# B&R Automation Studio project TD52 (part 133)

#### MsgSA.var
```iecst
VAR
	iAdrAmmBase2MM : UDINT;
	iAdrMM2AmmBase : UDINT;
	xMsg2214 : Msg;
	xMsg2254 : Msg;
	xMsg2255 : Msg;
	xMsg2256 : Msg;
	xMsg2281 : Msg;
	xMsg2297 : Msg;
	xMsg2298 : Msg;
	xMsg2299 : Msg; (* alarm for cylinder pressure sensor saturation*)
	xMsg9318 : Msg; (* warning for cylinder pressure sensor saturation*)
	xMsg2585 : Msg;
	xMsg2800 : Msg;
	xMsg2816 : Msg;
	xMsg2817 : Msg;
	xMsg2818 : Msg;
	xMsg2819 : Msg;
	xMsg2820 : Msg;
	xMsg2898 : Msg;
	xMsg2906 : Msg;
	xMsg2907 : Msg;
	xMsg3270 : Msg;
	xMsg3271 : Msg;
	xMsg3272 : Msg;
	xMsg3273 : Msg;
	xMsg3275 : Msg;
	xMsg3276 : Msg;
	xMsg3277 : Msg;
	xMsg3278 : Msg;
	xMsg3283 : Msg;
	xMsg3284 : Msg;
	xMsg3286 : Msg;
	xMsg3287 : Msg;
	xMsg3288 : Msg;
	xMsg3291 : Msg;
	xMsg3292 : Msg;
	xMsg3293 : Msg;
	xMsg3294 : Msg;
	xMsg3330 : Msg;
	xMsg3331 : Msg;
	xMsg3332 : Msg;
	xMsg3333 : Msg;
	xMsg3334 : Msg;
	xMsg3335 : Msg;
	xMsg3336 : Msg;
	xMsg3337 : Msg;
	xMsg3338 : Msg;
	xMsg3343 : Msg;
	xMsg3344 : Msg;
	xMsg3345 : Msg;
	xMsg3530 : Msg;
	xMsg3531 : Msg;
	xMsg3533 : Msg;
	xMsg3535 : Msg;
	xMsg3536 : Msg;
	xMsg3537 : Msg;
	xMsg3539 : Msg;
	xMsg3544 : Msg;
	xMsg3545 : Msg;
	xMsg3546 : Msg;
	xMsg3547 : Msg;
	xMsg3548 : Msg;
	xMsg3549 : Msg;
	xMsg3550 : Msg;
	xMsg3551 : Msg;
	xMsg3552 : Msg;
	xMsg3553 : Msg;
	xMsg3554 : Msg;
	xMsg2910 : Msg;
	xMsg2476 : Msg;
	xMsg2334 : Msg;
	xMsg9027 : Msg;
	xMsg2335 : Msg;
	xMsg9028 : Msg;
	xMsg9320 : Msg;
	xMsg9045 : Msg;
	xMsg9321 : Msg;
	xMsg9046 : Msg;
	xMsg2493 : Msg;
	xMsg2939 : Msg;
	xMsg9066 : Msg;
	xMsg9050 : Msg;
	xMsg9350 : Msg;
END_VAR
```


### Package Logical/Synchronization - SY: Synchronization

### Data object Logical/Synchronization/META_SY (Simple) - MODUL META data file

#### META_SY.dat
```
; *******************************************************************************
; AGGR: Module Meta Data (data module)
;
; This code is confidential and proprietary to the INNIO Company.
; It may not be used in any form, or reproduced in any manner, without the express
; written permission of the INNIO Company.
; Copyright, INNIO Company, 2022
;
; Customized modifications: -
; ------------------------
;
; History:
; -------
; V03.99.00.00	06.03.2013	Weitzer, 	generated for modular software
;				02.10.2013	lettenb.	descriptions setted
;				04.12.2013	lettenb.	dependencies added
; V04.00.00.00	31.01.2014	lettenb.	version + dependencies changed
; V04.00.03.00	22.07.2014	lettenb.	para_task update
; V04.03.00.00	02.03.2015	lettenb.	version + dependencies changed (920)
; V04.03.00.00	11.06.2015	Zengerer 	version + dependencies changed (IF change with array index 0 for compatibility with c-tasks)
;				15.06.2015  lettenb.	PARAMETER_CHK expanded
; V04.04.00.00	04.07.2016	lettenb.	version changed
;               20.03.2017  lettenb.	fast detection of freq.changes, dyn.gridcode III
; V04.05.00.00	11.12.2017	lettenb.	gridcode logic added
; V04.05.01.00	09.03.2018	Perktold	delayed A1042 trip (only HiHi part), 100ms normal, 500ms when LVRT Event is detected (for 5s)
;               18.09.2018	lettenb.	gcb IO monitoring, sequential arrangement changed, bu
; V04.06.00.00	21.09.2018  Perktold,   MsgSY: A1042 implemented 110% overload step 3s delay excluded bBDC_Emergency_OFF
; V04.07.00.00	11.12.2017	lettenb.	dataitems for diagnosis added
;				03.10.2019	lettenb.	perm data writing to CF 10s -> 10m, bu01
; V04.09.00.00	17.10.2019	lettenb.	gcbTC1, gcb closing time monitoring added
;				01.10.2020	lettenb.	OUT_SY.bMCB_DemSy, mcb controlled by customer, bugfix(heim, Referenzanlage AB85), bu02
; V04.10.00.00	16.10.2020  Weitzer		IN_SY.bCust_Dem_Sy added to GCB demand sy, IN_SY.bCust_Dem_RSy added to ton_mcb_dmnd_sy ELSE part
; V04.11.00.00	24.06.2021	Arnold		Open GCB in island on underfrequency IN_SY.bGCB_DCon_EC
;				07.07.2021	lettenb.	init xMsg2692.Num: 2693->2692, bugfix
; V04.12.00.00	02.05.2022	Schmidt		W2688 (high sync current) threshold increased from 50% to 75% of nominal current
;				29.06.2022	lettenb.	dead bb synch added
; V04.13.00.00  26.09.2023	Farre,		LCB operating message when open (B9083) or closed (B9084)
;				14.11.2023	Hohensinner	Added LV_GCB task (Modbus RTU connection to LV GCBs)
;				20.11.2023	Farre,		added "bypass MCB" and "request power mode" interfaces from CU needed for Microgrid (2023-168)
;				29.11.2023	Goenczi,	Standardization changes (Aggreko)
;				22.01.2024	Astner		Added iModule to OUT_SY
; V04.14.00.00	25.10.2024	Farre,		GCB Opening Failure - W1217 and reverse power connected to GCB_OpF command (2024-241)
;				22.11.2024	Fahringer	Use generator current before GCB closure to check 2% change (2024-238)
;										GCB closing time monitoring for more than 40ms (2024-238)
;				22.11.2024	Farre		bMMD_SyncDO only when used for GCB (2024-238)
;
; Instructions for use:
; --------------------
; make only changes at the version numbers
;
; Outstandings:
; ------------
;
; *******************************************************************************
;
"<META>"
;
; Module ID
"<MODUL>SY</MODUL>"
;
; Module Version (xx.yy.zz.cc)
"<VERSION>04.14.00.00</VERSION>"
;
; Module Basisupdate Version BU (00-99)
"<BASISUPDATE_VERSION>00</BASISUPDATE_VERSION>"
;
; Optional: specify order number for limitated module usage
"<ORDER></ORDER>" ;<!--(optional for restricted customizations; missing statement makes module valid for all orders)-->
;
; Parameter Check <PARAn Name='aAbcdef' MIN='xxx' MAX='yyy' />  (watch for correct spacings and apostrophs!)
"<PARAMETER_CHK>"
"<PARA1 Name='iEng_Motortype' MIN='208' MAX='920' />"
"<PARA2 Name='rN_EngStart_LimHi' MIN='50.0' MAX='2200.0' />"
"<PARA3 />"
"<PARA4 />"
"<PARA5 />"
"</PARAMETER_CHK>"
;
; Permanent Datamodule Filenames<!-- NAME ist ohne Dateiendung einzutragen; Nur für Counter und interne Parameter verwenden-->
"<DATAMODULES>" ;<!-- optional; mehrere DATAMODULES erlaubt-->
"	<DATAMODULE>par_SY</DATAMODULE>"
"	<DATAMODULE>perm_SY</DATAMODULE>"
"</DATAMODULES>"
;
; Dependencies Modules (MMxx.yy.zz.cc)
"<DEPENDENCIES>"
"	<DEPENDENCY MODULE='AB' VERSION='04.03.00.00' />"
"	<DEPENDENCY MODULE='CH' VERSION='04.00.00.00' />"
"	<DEPENDENCY MODULE='CU' VERSION='04.13.00.00' />"
"	<DEPENDENCY MODULE='EC' VERSION='04.06.00.00' />"
"	<DEPENDENCY MODULE='EG' VERSION='04.00.00.00' />"
"	<DEPENDENCY MODULE='GC' VERSION='04.14.00.00' />"
"	<DEPENDENCY MODULE='GR' VERSION='04.07.00.00' />"
"	<DEPENDENCY MODULE='GT' VERSION='04.00.00.00' />"
"	<DEPENDENCY MODULE='HA' VERSION='04.13.00.00' />"
"	<DEPENDENCY MODULE='HC' VERSION='04.07.00.00' />"
"	<DEPENDENCY MODULE='IG' VERSION='04.00.00.00' />"
"	<DEPENDENCY MODULE='OP' VERSION='04.13.00.00' />"
"	<DEPENDENCY MODULE='PB' VERSION='04.00.00.00' />"
"   <DEPENDENCY VISVERSION='02.14.00.00' />"			; Dependencies Visualization
"</DEPENDENCIES>"
;
; Module function description
"<MODULEFUNCTION>" ;<!-- short overview documentation of module function; add reference to detailed information, if available-->
"	<General>	"
"	Circuit breaker control. "
"	</General>	"
""
"	<F1 Name='Generator circuit breaker' LastModified='3.99.00.00'>"
"	Generator circuit breaker control and monitoring.	"
"	</F1>"
"	<F2 Name='Mains circuit breaker' LastModified='3.99.00.00'>"
"	Mains circuit breaker control and monitoring.	"
"	</F2>"
"	<F3 Name='Blackout start' LastModified='3.99.00.00'>"
"	Blackout start management.	"
"	</F3>"
"	<F4 Name='Load shedding' LastModified='3.99.00.00'>"
"	Load shedd management.	"
"	</F4>"
"	<F5 Name='Generator deexcitation' LastModified='3.99.00.00'>"
"	Generator deexcitation control.	"
"	</F5>"
"	<F6 Name='Synchronization alarm management' LastModified='4.04.00.00'>"
"	Synchronization alarm management.	"
"	</F6>"
"	<F7 Name='Mains monitoring' LastModified='4.04.00.00'>"
"	Mains monitoring (dyn.gridcode III)"
"	</F7>"
""
"	<Info>"
"   UPDATE V4.02.01	version + dependencies changed (IF change with array index 0 for compatibility with c-tasks)	"
"	</Info>"
""
"	<Customized LastModified='3.99.00.00'>"
"	- Nothing "
"	</Customized>	"
""
"</MODULEFUNCTION>"
;
"</META>"
```

### module_SY.typ
```iecst
TYPE
	IN_SY_struct : 	STRUCT
		tAB2SY : AmmBase2MM;
		tPB2MM : ParaBase2MM_type;
		iSt_OpMode : UDINT; (*status operation mode*) (*OldName:newPv; Cycle:5;*)
		iIdx_OMSS : INT; (*engine operation mode selection*) (*OldName:newPv; Cycle:5;*)
		rN_EngAct : REAL; (*engine speed actual [1/min]*) (*OldName:ANA.DREHZ; Cycle:5;*)
		bEng_RPSDem : BOOL; (*engine demanded *) (*OldName:A_AGFD; Cycle:5;*)
		bEng_Rdy_Aut_Exc : BOOL; (* engine ready for automatic operation *) (*OldName:BERAUT; Cycle:5;*)
		bGCB_Off_CNS : BOOL; (* generator circuit breaker opened by curent negative sequence *) (*OldName:gcb_off_iasy; Cycle:5;*)
		bGCB_Off_RP : BOOL; (* generator circuit breaker opened by reverse power *) (*OldName:gcb_off_rlsg; Cycle:5;*)
		bEng_Dem : BOOL; (* demand engine *) (*OldName:M_AGFD; Cycle:5;*)
		bEng_Dem_EPS : BOOL; (* engine demand for emergency operation *) (*OldName:M_NANF; Cycle:5;*)
		bGV_On : BOOL; (*Gas valves On *) (* OldName:M_GASV; Cyclic:5;*)
		rP_Nom : REAL; (* nominal power related to selected gas type [kW]*) (*OldName:PN_GASART[]; Cycle:5;*)
		bSCO_Active : BOOL; (* safety cut out gas valves glow ignition prevention *) (*OldName:SICH_SCHL; Cycle:5;*)
		rP_Act_Norm : REAL; (* actual power related to rP_Nom [%] *) (*OldName:P_IST_OF; Cycle:5;*)
		rP_Act_Norm_Filt : REAL; (* actual power related to rP_Nom filtered(1s) [%] *) (*OldName:P_IST; Cycle:5;*)
		bP_Red_Active : BOOL; (* power reduction active - any kind *) (*OldName:PredAkt; Cycle:5;*)
		bRelSy_Customized : BOOL; (*release synchronization from custom)*) (*OldName:newPv; Cycle:5;*)
		rP_MainsImport : REAL; (* mains import power [kW]*) (*OldName:Pmns_pv_1; Cycle:5;*)
		tEng_Run : HALioDo_Type; (* engine in operation *) (*OldName:BTRB; Cycle:5;*)
		tRel_Sync_Load : HALioDo_Type; (*DO release of sychronization and load*) (*OldName:SY_LFG; Cycle:5;*)
		tGrC_DCon : HALioDo_Type; (*DO: FALSE = Disconnect from Grid due to GridCode Event*) (* OldName: DO_GRIDCODE_DCON_TC1; Cycle:5; *)
		tTBMode : HALioDi_Type; (* DI test bench mode *) (*OldName:CIRCUITUS; Cycle:5;*)
		tBB_Alive : HALioDi_Type; (* DI bus bar alive *) (*OldName:DI_BB_ALIVE; Cycle:5;*)
		tBB_Dead_MMD : ARRAY[0..2]OF HALioDi_Type; (* DI bus bar dead from MMD *) (*OldName:DI_MMUSynchStatDO03; Cycle:5;*)
		tC_CB_EDC : HALioDi_Type; (* DI customer circuit breaker (engine) demand close *) (*OldName:DI_C_CB_EDC; Cycle:5;*)
		tC_CB_ESL : HALioDi_Type; (* DI customer circuit breaker (engine) status locked *) (*OldName:DI_C_CB_ESL; Cycle:5;*)
		tC_CB_Off : HALioDi_Type; (* DI customer circuit breaker opened *) (*OldName:DI_C_CB_OFF; Cycle:5;*)
		tC_CB_On : HALioDi_Type; (* DI customer circuit breaker closed *) (*OldName:DI_C_CB_ON; Cycle:5;*)
		tReq_PowMod : HALioDi_Type; (* DI request power operation mode *) (*OldName:DI_DMND_PM; Cycle:5;*)
		tEngDemIsland : HALioDi_Type; (* DI engine demand for island operation *) (*OldName:DI_ENG_DI; Cycle:5;*)
		tGCB_AGO : HALioDi_Type; (* DI all other generator circuit breaker off *) (*OldName:DI_GCB_AGO; Cycle:5;*)
		tGCB_DSY : HALioDi_Type; (* DI  generator circuit breaker demand synchronization (synchline) *) (*OldName:DI_GCB_DSY; Cycle:5;*)
		tGCB_DVM : HALioDi_Type; (* DI  generator circuit breaker demand voltage matching *) (*OldName:DI_GCB_DVM; Cycle:5;*)
		tGCB_MDL : HALioDi_Type; (* DI generator circuit breaker master demand lock (for closing other GCB to dead BB) *) (*OldName:DI_GCB_MDL; Cycle:5;*)
		tGCB_MRC : HALioDi_Type; (* DI generator circuit breaker master release close (to dead busbar) *) (*OldName:DI_GCB_MRC; Cycle:5;*)
		tGCB_OGP : HALioDi_Type; (* DI generator circuit breaker other generator parallel *) (*OldName:DI_GCB_OGP; Cycle:5;*)
		tGCB_On : HALioDi_Type; (* DI generator circuit breaker closed *) (*OldName:DI_GCB_ON; Cycle:5;*)
		tGCB_Rac : HALioDi_Type; (* DI generator circuit breaker racked in *) (*OldName:DI_GCB_RAC; Cycle:5;*)
		tGCB_Rdy : HALioDi_Type; (* DI generator circuit breaker ready (for close) *) (*OldName:DI_GCB_RDY; Cycle:5;*)
		tGCB_RI : HALioDi_Type; (* DI generator circuit breaker reelase island *) (*OldName:DI_GCB_RI; Cycle:5;*)
		tGCB_SM1 : HALioDi_Type; (* DI generator circuit breaker output signal monitoring 1 *) (*OldName:DI_GCB_SM1; Cycle:5;*)
		tGCB_SM2 : HALioDi_Type; (* DI generator circuit breaker contact signal monitoring 2 *) (*OldName:DI_GCB_SM2; Cycle:5;*)
		tGCB_Off : HALioDi_Type; (* DI generator circuit breaker opened *) (*OldName:DI_GCB_OFF; Cycle:5;*)
		tGCB_Earth : HALioDi_Type; (* DI generator circuit breaker position earth *) (*OldName:newPv; Cycle:5;*)
		tMCB_OL : HALioDi_Type; (* DI mains circuit breaker overload *) (*OldName:DI_MCB_OL; Cycle:5;*)
		tMCB_On : HALioDi_Type; (* DI mains circuit breaker closed *) (*OldName:DI_MCB_ON; Cycle:5;*)
		tMCB_Off : HALioDi_Type; (* DI mains circuit breaker opened *) (*OldName:DI_MCB_OFF; Cycle:5;*)
		tMCB_Rac : HALioDi_Type; (* DI mains circuit breaker racked in *) (*OldName:DI_MCB_RAC; Cycle:5;*)
		tMCB_Rdy : HALioDi_Type; (* DI mains circuit breaker ready (for close) *) (*OldName:DI_MCB_RDY; Cycle:5;*)
		tMCB_Rem : HALioDi_Type; (* DI mains circuit breaker remote (operating mode) *) (*OldName:DI_MCB_REM; Cycle:5;*)
		tMCB_SM : HALioDi_Type; (* DI mains circuit breaker signal monitoring *) (*OldName:DI_MCB_SM; Cycle:5;*)
		tMns_MDF : HALioDi_Type; (* DI mains monitoring device failure *) (*OldName:DI_MCB_MDF; Cycle:5;*)
		tMnsOk : HALioDi_Type; (* DI mains ok *) (*OldName:DI_MNS_OK; Cycle:5;*)
		tOnly_Island : HALioDi_Type; (* DI only island operation *) (*OldName:DI_ONLY_I; Cycle:5;*)
		tRel_BS : HALioDi_Type; (* DI release black start *) (*OldName:DI_REL_BS; Cycle:5;*)
		tRel_I : HALioDi_Type; (* DI release island operation *) (*OldName:DI_REL_I; Cycle:5;*)
		tRel_LS : HALioDi_Type; (* DI release load shedding *) (*OldName:DI_REL_LS; Cycle:5;*)
		tGCB_DRM : HALioDi_Type; (* DI generator circuit breaker demand MCB closing return to mains *) (*OldName:newPv; Cycle:5;*)
		tGen_RVM : HALioDi_Type; (* DI generator release voltage matching (leroy somer) *) (*OldName:newPv; Cycle:5;*)
		tSy_N_Up : HALioDi_Type; (* DI external speed matching UP *) (*OldName:newPv; Cycle:5;*)
		tSy_N_Down : HALioDi_Type; (* DI external speed matching DOWN *) (*OldName:newPv; Cycle:5;*)
		tLineCB_On : HALioDi_Type; (* DI line circuit breaker closed *) (*OldName:LIN_EIN; Cycle:5;*)
		tU_Avg : ARRAY[0..2]OF HALioAi_Type; (*AI generator voltage average value MMD [V]*) (*OldName:ANA.UDURCH; Cycle:5;*)
		tRelEngOpFromGSy : HALioDi_Type; (*DI release engine operation from 'gemeinsame'synchronization*) (*OldName:F_BLO; Cycle:5;*)
		tEarthCB_Off : HALioDi_Type; (*DI earth circuit breaker opened, france country specific*) (*OldName:DI_ECB_OFF; Cycle:5;*)
		tIsoCB_Off : HALioDi_Type; (*DI disconnecting circuit breaker opened, france country specific*) (*OldName:DI_ISOL; Cycle:5;*)
		tMnsOk_GTE : HALioDi_Type; (*DI mains ok GTE monitoring device, france country specific*) (*OldName:DI_GTE; Cycle:5;*)
		tMnsOk_TGS : HALioDi_Type; (*DI mains ok TGS monitoring device, france country specific*) (*OldName:DI_TGS; Cycle:5;*)
		tMnsOk_C13100 : HALioDi_Type; (*DI mains ok C13.100 monitoring device, france country specific*) (*OldName:DI_C13_100; Cycle:5;*)
		bMsg1026 : BOOL; (*engine shutdown failure *) (*OldName:M_ANSTAB; Cycle:5;*)
		bMsg1026_Test : BOOL; (*engine shutdown failure test*) (*OldName:newPv; Cycle:5;*)
		bMsg1134 : BOOL; (*Earth failure*) (*OldName:M_ERDS; Cycle:5;*)
		bMsg1036 : BOOL; (*overload short circuit*) (*OldName:M_ULKS; Cycle:5;*)
		bMsg1038 : BOOL; (*generator reverse power*) (*OldName:M_RLSG; Cycle:5;*)
		bMsg1073 : BOOL; (*generator over load from multi measuring device*) (*OldName:M_MMD_OL; Cycle:5;*)
		bMsg1132 : BOOL; (*generator differencial protection*) (*OldName:M_DIFF; Cycle:5;*)
		bMsg3319 : BOOL; (*generator protection trip*) (*OldName:M_GEN_PT; Cycle:5;*)
		rCust_SparePara : ARRAY[0..200]OF REAL; (*SPS_REZP1 to SPS_REZP200	*) (* OldName: SPS_REZP1, SPS_REZP2, SPS_REZP70; Cycle: 5; *)
		tCustAnaIn : ARRAY[0..120]OF HALioAi_Type; (*Replacement for RAN_KANAL...*) (*OldName: ANA_RAN	; Cycle: 5;*)
		tCustDigIn : ARRAY[0..200]OF HALioDi_Type; (*new, reserved for Project specific use*) (*OldName: new PV	; Cycle: 5;*)
		tMCB_Rel_Sync_SOn : HALioDo_Type; (* DO: releas decoupling quickly from EU (ERDF) *) (*OldName:DO_RMFrgKop ;Cycle:5;*)
		bServiceMode : BOOL; (*service mode*) (*OldName:bServiceBegin; Cycle:5;*)
		bBDC_Emergency_OFF : BOOL; (*over load - emergency off*) (*OldName:new PV; Cycle:5;*)
		tPr_Ch_P2s : HALioAi_Type; (*actual charge pressure before throttle valve(P2s)[bar]*) (*OldName:pl_ist; Cycle:5;*)
		tPr_Ch_P2s_A : HALioAi_Type; (*actual charge pressure before throttle valve(P2s)bank A[bar]*) (*OldName:pl_ist; Cycle:5;*)
		tPr_Ch_P2s_B : HALioAi_Type; (*actual charge pressure before throttle valve(P2s)bank B[bar]*) (*OldName:pl_ist; Cycle:5;*)
		tMnsOk_ClosCond_Ok : HALioDi_Type; (*closing condition from external facility*) (*OldName:newPV; Cycle:5*)
		tU_MMD_Synch2 : ARRAY[0..2]OF HALioAi_Type; (*phase voltage system 2*) (*OldName:ssSynch2Volt; Cycle:5*)
		tF_MMD_Synch2 : ARRAY[0..2]OF HALioAi_Type; (*frequency sync-system 2*) (*OldName:usSynch2Frequency; Cycle:2*)
		iIdx_Eng_State : INT; (* state of engine *) (*OldName:HPTSCHL; Cycle:5;*)
		tMCB_OpF_Ext : HALioDi_Type; (*generator circuit breaker opening failure*) (*OldName:newPV; Cycle:5*)
		tGCB_OpF_Ext : HALioDi_Type; (*generator circuit breaker opening failure*) (*OldName:newPV; Cycle:5*)
		tTempMax_GenCB : HALioDi_Type; (*Temperature max generator switch gear*)
		bEng_Bloc : BOOL; (* blocking engine *) (*OldName:M_BLOCK;Cycle:5;*)
		bMMD_GenAlarmTestOn : BOOL; (*MMD_Gen alarm test On*) (*OldName:newPv; Cycle:5;*)
		bMMD_BB_AlarmTestOn : BOOL; (*MMD_BB  alarm test On*) (*OldName:newPv; Cycle:5;*)
		rI_MaxL1 : ARRAY[0..2]OF REAL; (* max. generator current phase 1 [A]  *) (* OldName:ssIMaxL1; Cycle: *)
		rI_MaxL2 : ARRAY[0..2]OF REAL; (* max. generator current phase 2 [A]  *) (* OldName:ssIMaxL2; Cycle: *)
		rI_MaxL3 : ARRAY[0..2]OF REAL; (* max. generator current phase 3 [A]  *) (* OldName:ssIMaxL3; Cycle: *)
		bType6_Update_Rel : BOOL; (* Enables Type6 Engine controls Update (100% Loadrejection, Island mode etc..) *) (*OldName:newPv; Cycle:5;*)
		bT_ECW_Lo : BOOL; (*temperature engine cooling water limit low*) (*OldName:AN_KTMI; Cycle:5;*)
		tU_Bus_L3_1 : ARRAY[0..2]OF HALioAi_Type; (* Line voltage bus bar 3 1 *) (*OldName:ssBusVoltPh3_1; Cycle:5*)
		tU_Bus_L2_3 : ARRAY[0..2]OF HALioAi_Type; (* Line voltage bus bar 2 3 *) (*OldName:ssBusVoltPh2_3; Cycle:5*)
		tU_Bus_L1_2 : ARRAY[0..2]OF HALioAi_Type; (* Line voltage bus bar 1 2 *) (*OldName:ssBusVoltPh1_2; Cycle:5*)
		bGridCode_ON : BOOL; (*any dyn. GridCode function activated*)
		bGen2_Act : BOOL; (* TRUE = Gen2 Controller active*) (* Oldname: BDC_ON; Cycle: 2 *)
		tMnsOk_ClosCond_Skip : HALioDi_Type; (*skip closing condition from external facility*) (* OldName: newPV; Cycle:5; *)
		tAfMnsF_ClosCond_Ok : HALioDi_Type; (*closing condition from external facility after mains failure*) (* OldName: newPV; Cycle:5; *)
		tAfMnsF_ClosCond_Skip : HALioDi_Type; (*skip closing condition from external facility after mains failure*) (* OldName: newPV; Cycle:5; *)
		tHW_Switches : OpMode_Switches; (*Hardware operation mode switches*)
		tF_MMD_BusBar : ARRAY[0..2]OF HALioAi_Type; (*frequency busbar*) (*OldName:usSynch2Frequency; Cycle:2*)
		bTP_GrC_Event : BOOL; (* Grid Code Event*) (*OldName: bGridCodeEvent;*)
		tMidVoltCB_Failure : HALioDi_Type; (*mid voltage CB failure*)
		tAuxV_Supply_Ok : HALioDi_Type; (*DI auxiliary voltage supply ok*) (*OldName:SPG_HBT; Cycle:5;*)
		bDem_I_Bus : BOOL; (* Demand Island Operation by Bus *)
		bRel_I_Bus : BOOL; (* Release Island Operation by Bus *)
		bDem_Sy_Bus : BOOL; (* Demand synchronization by Bus *)
		bDem_RSy_Bus : BOOL; (* Demand re-synchronization by Bus *)
		bDem_BS_GCBOn_Bus : BOOL; (* Demand blouck-out start with GCB closed by Bus *)
		bDem_BS_DeExc_Bus : BOOL; (* Demand blouck-out start with deexcitation by Bus *)
		bGCB_by_Customer : BOOL; (* GCB controled by Customer *)
		bMMD_SynchDO : ARRAY[0..2]OF BOOL; (* feedback synch DO *) (* OldName:new PV;*)
		bMMD_SynchDO_TC1 : ARRAY[0..2]OF BOOL; (* feedback synch DO *) (* OldName:new PV;*)
		tI_L1_TC1 : ARRAY[0..2]OF HALioAi_Type; (*Phase current generator I1 *) (*OldName:ssIL1_fast;*)
		tI_L2_TC1 : ARRAY[0..2]OF HALioAi_Type; (*Phase current generator I2 *) (*OldName:ssIL2_fast;*)
		tI_L3_TC1 : ARRAY[0..2]OF HALioAi_Type; (*Phase current generator I3 *) (*OldName:ssIL3_fast;*)
		bCust_Dem_Sy : BOOL; (* Demand synchronization from CU module *) (*OldName:ssBusVoltPh1_2; Cycle:5*)
		bCust_Dem_RSy : BOOL; (* Demand re-synchronization from CU module *) (*OldName:ssBusVoltPh1_2; Cycle:5*)
		tGndFault_BB : HALioDi_Type; (*earth fault bus bar*)
		bGCB_DCon_EC : BOOL; (*GCB open command from EngineController *)
		tDemGenExcOff : HALioDi_Type; (*demand generator excitation off*)
		bBypassMCB_deadBB : BOOL; (*bypass MCB status information from the standard dead_bb check*)
		bBypassMCB_SoftStart : BOOL; (*bypass MCB status information from the standard soft energisation logic*)
		bBypassMCB_LoadShed : BOOL; (*bypass MCB status information from the standard load shedding logic*)
		bSoftEnergDem : BOOL; (*demand transformer soft energisation*)
		bReq_PowMod : BOOL; (*request power mode - over-written in customization*)
		bCust_Rel_I : BOOL; (*release island from CU module*)
		bCust_RelI_BB : BOOL; (*release VKE10 from CU module (Aggreko)*)
		bCust_Dem_EPS_Sy : BOOL; (*demand EPS from CU module*)
		bSmoothDischarge_CU : BOOL; (*Smooth engine discharge in Island mode set in CU*)
		bSetGCB2Close : BOOL; (*External GCB close command*)
		bSetGCB2Open : BOOL; (*External GCB open command*)
		bSetFixedPwrMode : BOOL; (*Set power mode event based*)
		bOM_Bus : BOOL; (*Operation mode via BUS*) (*OldName:OperationModeModbus; Cycle:5;*)
		bSetIslandMode : BOOL; (*Set island mode event based*)
		bSetAutControlMode : BOOL; (*Set manual conrol mode event based *)
		bSetManControlMode : BOOL; (*Set auto conrol mode event based*)
		bBus_Active : BOOL; (*Bus communication active*) (*OldName:Modbus_activ; Cycle:5;*)
		bGCB_OGP_Bus : BOOL; (* other generator parallel over Modbus*)
		bPact_Rev : BOOL; (*reverse power*)
	END_STRUCT;
END_TYPE

(*END_IN*)

TYPE
	OUT_SY_struct : 	STRUCT
		tIsland_Op : HALioDo_Type; (*Island operation*) (*OldName:A_USP; Cycle:5;*)
		tParallel_Op : HALioDo_Type; (*mains parallel operation*) (*OldName:A_USP; Cycle:5;*)
		tSY2AB : MM2AmmBase;
		tSY2PB : MM2ParaBase_type;
		bSyncSlipMode : ARRAY[0..2]OF BOOL; (*MMD synchronization with slip mode*) (*OldName:bSyncSlipMode; Cycle:5;*)
		bEng_Dem_EPS_Sy : BOOL; (*engine demand emergency power supply from synch.*) (*OldName:ANF_NSB; Cycle:5;*)
		bMCB_DemSy : BOOL; (* demand synchronization mains circuit breaker *) (*OldName:ARSYANW,mcb[1].dmnd_sy; Cycle:5;*)
		bGCB_DemSy : BOOL; (* demand synchronization generator circuit breaker *) (*OldName:ASYANW,gcb[1].dmnd_sy; Cycle:5;*)
		bGen_SyD_Dem : BOOL; (* demand synch.device *) (*OldName:dmnd_sy_device; Cycle:5;*)
		bRelEngOpFromSy : BOOL; (* release engine operation from synchronization *) (*OldName:M_FBLO; Cycle:5;*)
		bRel_Island : BOOL; (* release island operation *) (*OldName:FG_INSEL; Cycle:5;*)
		bDSyLine : BOOL; (* demand synchline *) (*OldName:M_SYL; Cycle:5;*)
		bMCB_On : BOOL; (* mains circuit breaker closed *) (*OldName:MCB_ON; Cycle:5;*)
		bMnsOk : BOOL; (* mains ok *) (*OldName:NE_OK; Cycle:5;*)
		bMainsReturn : BOOL; (* mains return *) (*OldName:NWK; Cycle:5;*)
		bOtherGenParallel : BOOL; (* other generator parallel *) (*OldName:PARALLEL; Cycle:5;*)
		bOnly_Island : BOOL; (* only island operation *) (*OldName:REIN_INSEL; Cycle:5;*)
		bMsg1218 : BOOL; (* generator circuit breaker opening failure *) (*OldName:S_AUS_GS; Cycle:5;*)
		bMsg1219 : BOOL; (* generator circuit breaker closing failure *) (*OldName:S_EIN_GS; Cycle:5;*)
		bMsg1217 : BOOL; (* generator circuit breaker position signal failure *) (*OldName:S_STL_GS; Cycle:5;*)
		bMsg1209 : BOOL; (* mains circuit breaker position signal failure *) (*OldName:S_STL_NS; Cycle:5;*)
		bSmoothDischarge : BOOL; (* smooth engine discharge *) (*OldName:SANFT; Cycle:5;*)
		bBB_dead : BOOL; (* bus bar dead *) (*OldName:SS_OSP; Cycle:5;*)
		bSynchDem : BOOL; (* synchronization demanded *) (*OldName:SynchAnf; Cycle:5;*)
		bGen_Exc_Off : BOOL; (* de- excitation *) (*OldName:T_ENTR; Cycle:5;*)
		bRel_IslandAfMITime : BOOL; (* jump release island op.after mi-filter time *) (*OldName:T79; Cycle:5;*)
		bTestBenchModeIsland : BOOL; (* test bench mode - island mode *) (*OldName:PRF_I; Cycle:5;*)
		bTestBenchModeParallel : BOOL; (* test bench mode - parallel mode *) (*OldName:PRF_NP; Cycle:5;*)
		tGCB_RUC : HALioDo_Type; (* generator circuit breaker release undervoltage coil *) (*OldName:A_USP; Cycle:5;*)
		tGCB_COf : HALioDo_Type; (* command gcb off *) (*OldName:DO_GCB_COF; Cycle:5;*)
		tMCB_COf : HALioDo_Type; (* command mcb off *) (*OldName:DO_MCB_COF; Cycle:5;*)
		tDemandBB : HALioDo_Type; (* demand busbar *) (*OldName:DO_DMND_BB; Cycle:5;*)
		tEng_Dem : HALioDo_Type; (* engine demanded for MSY *) (*OldName:DO_ENG_D; Cycle:5;*)
		tEng_Run_Sy : HALioDo_Type; (* engine runing - synchronization*) (*OldName:DO_ENG_RUN; Cycle:5;*)
		tGCB_COn : HALioDo_Type; (* command gcb on *) (*OldName:DO_GCB_CON; Cycle:5;*)
		tGCB_DVS : HALioDo_Type; (* generator circuit breaker demand voltage selection *) (*OldName:DO_GCB_DVS; Cycle:5;*)
		tGCB_EDC : HALioDo_Type; (* generator circuit breaker engine demand close  *) (*OldName:DO_GCB_EDC; Cycle:5;*)
		tGCB_ESL : HALioDo_Type; (* generator circuit breaker status locked  *) (*OldName:DO_GCB_ESL; Cycle:5;*)
		tGCB_OpF : HALioDo_Type; (* generator circuit breaker opening failure  *) (*OldName:DO_GCB_OPF; Cycle:5;*)
		tGCB_Rel : HALioDo_Type; (* generator circuit breaker release closing  *) (*OldName:DO_GCB_REL; Cycle:5;*)
		tGCB_RSP : HALioDo_Type; (* generator circuit breaker release synch pulse  *) (*OldName:DO_GCB_RSP; Cycle:5;*)
		tGCB_RT : HALioDo_Type; (* generator circuit breaker release trip  *) (*OldName:DO_GCB_RT; Cycle:5;*)
		tLock_C_MCB : HALioDo_Type; (* lock customer mains circuit breaker *) (*OldName:DO_LOCK_C_MCB; Cycle:5;*)
		tMCB_COn : HALioDo_Type; (* mains circuit breaker comand on *) (*OldName:DO_MCB_CON; Cycle:5;*)
		tMCB_DVS : HALioDo_Type; (* mains circuit breaker demand voltage selection *) (*OldName:DO_MCB_DVS; Cycle:5;*)
		tMCB_RSP : HALioDo_Type; (* mains circuit breaker release synch pulse  *) (*OldName:DO_MCB_RSP; Cycle:5;*)
		tMCB_RT : HALioDo_Type; (* mains circuit breaker release trip  *) (*OldName:DO_MCB_RT; Cycle:5;*)
		tPulseMainsOk : HALioDo_Type; (* pulse mains ok *) (*OldName:DO_PUL_MNS_OK; Cycle:5;*)
		tRdy_MSy : HALioDo_Type; (* engine ready for MSY *) (*OldName:DO_RDY_MSY; Cycle:5;*)
		tGenDeexitDem : HALioDo_Type; (* DO generator deexitation demand *) (*OldName:A_ENTR; Cycle:5;*)
		tP_Lo : HALioDo_Type; (* DO power low (for opening GCB) *) (*OldName:P_MIN; Cycle:5;*)
		tN_EngStart : HALioDo_Type; (* DO engine startup speed exceeded*) (*OldName:A_DREHZ; Cycle:5;*)
		tLS_Dem : HALioDo_Type; (*DO load shedding demand*) (*OldName:DO_DMND_LS; Cycle:5;*)
		iIdx_SyOMSS : INT; (*synchronization operating mode selection*) (*OldName:newPv; Cycle:5;*)
		bRelMainsConnect : BOOL; (*Blocking module*) (*OldName:newPv; Cycle:5;*)
		tMCB_COf_GCB_OpF : HALioDo_Type; (*DO opening MCB in case of GCB opening failure*) (*OldName:newPv; Cycle:5;*)
		rP_Red_TempMax_GenCB_Norm : REAL; (*Setpoint power reduction temperature max generator switch gear*) (*OldName:newPv; Cycle:5;*)
		bP_Red_TempMax_GenCB_Sel : BOOL; (*Set power reduction temperature max generator switch gear*) (*OldName:newPv; Cycle:5;*)
		tLockEng_ClosCond : HALioDo_Type; (*lock engine due to closing conditions*) (*OldName:newPv; Cycle:5;*)
		tOMSS_Man : HALioDo_Type; (*operating mode selection man*) (*OldName:BWS_H; Cycle:5;*)
		tOMSS_Aut : HALioDo_Type; (*operating mode selection aut*) (*OldName:BWS_A; Cycle:5;*)
		tClosCond : HALioDo_Type; (*closing conditions ok*) (*OldName:newPv; Cycle:5;*)
		tAfMnsF_ClosCond : HALioDo_Type; (*closing conditions ok after mains failure*) (*OldName:newPv; Cycle:5;*)
		tAfMnsF_LockEng_ClosCond : HALioDo_Type; (*lockout engine due to closing conditions after mains failure*) (*OldName:newPV; Cycle:5;*)
		bSel_DeExc : BOOL; (* Deexcitation selected *)
		bGen_DeExc_Rdy : BOOL; (* Generator Deexitation ready *)
		bMsg1041Set : BOOL; (*power signal missing*)
		bMsg1042Set : BOOL; (*power signal overload*)
		bMsg2801Set : BOOL; (*module blocked by grid connection conditions*)
		bMsg2934Set : BOOL; (*module blocked by grid connection conditions after mains failure*)
		tGenExcOff : HALioDo_Type; (*generator de-energized(excitation off)*)
		tSyOMSS_Man : HALioDo_Type; (*synchronization operating mode selection MANUAL*)
		tSyOMSS_Aut : HALioDo_Type; (*synchronization operating mode selection AUTO*)
		bGCB_aut_on2dead_bb : BOOL; (*generator circuit breaker automatic on to dead bus bar*)
		iModule : USINT; (*Engine Module Number*)
		bGCB_psf_EngStop : BOOL; (*gcb position failure when engine stopped*)
	END_STRUCT;
END_TYPE

(*END_OUT*)

TYPE
	MM2VIS_Struct : 	STRUCT
		bMnsOk : BOOL; (*mains ok*) (*OldName:B_SV[7]; Cycle:5;*)
		bNotMainsReturn : BOOL; (*not mains return*) (*OldName:RPMZ1; Cycle:5;*)
		bGCB_On : BOOL; (*gcb closed for report time measuring*) (*OldName:B_SV[11]; Cycle:5;*)
		bGCB_GnlWarning : BOOL; (* gcb general failure *) (*OldName:B_SV[8]; Cycle:5;*)
		bDSyGCB : BOOL; (*demand synchronization gcb*) (*OldName:B_SV[10]; Cycle:5;*)
		bMCB_On : BOOL; (*mcb closed for report time measuring*) (*OldName:B_SV[19]; Cycle:5;*)
		bMCB_GnlWarning : BOOL; (*mcb general failure*) (*OldName:B_SV[16]; Cycle:5;*)
		bDSyMCB : BOOL; (*demand synchronization gcb*) (*OldName:B_SV[18]; Cycle:5;*)
		bEngDemIsland : BOOL; (* DI engine demand for island operation *)
		bOnly_Island : BOOL; (* DI only island operation *)
		bGCB_MDL : BOOL; (* DI generator circuit breaker master demand lock (for closing other GCB to dead BB) *)
		bGCB_MRC : BOOL; (* DI generator circuit breaker master release close (to dead busbar) *)
		bGCB_AGO : BOOL; (* DI all other generator circuit breaker off *)
		bGCB_RI : BOOL; (* DI generator circuit breaker reelase island *)
		bGCB_OGP : BOOL; (* DI generator circuit breaker other generator parallel *)
		bGCB_DVM : BOOL; (* DI all other generator circuit breaker off *)
		bGCB_DSY : BOOL; (* DI generator circuit breaker demand synchronization (synchline) *)
		bRdy_MSy : BOOL; (* DO engine ready    for MSY/GSY *)
		bEng_Run_Sy : BOOL; (* DO engine rotating for MSY/GSY *)
		bEng_Dem : BOOL; (* DO engine demanded for MSY/GSY *)
		bGCB_OpF : BOOL; (* DO alarm gcb opening failure *)
		bGCB_EDC : BOOL; (* DO ESY demand lock all other cb's connected to dead busbar *)
		bGCB_ESL : BOOL; (* DO ESY status gcb locked *)
		bMsg1038 : BOOL; (*Generator reserve power*) (*OldName:newPV; Cycle:5;*)
		bMsg1039 : BOOL; (*synchronizing failure (time out)*) (*OldName:AMM_A10xx[]; Cycle:5;*)
		bMsg1041 : BOOL; (*power signal missing*) (*OldName:AMM_A10xx[]; Cycle:5;*)
		bMsg1042 : BOOL; (*power signal overload*) (*OldName:AMM_A10xx[]; Cycle:5;*)
		bMsg1109 : BOOL; (*Generator loss of excitation*) (*OldName:newPV; Cycle:5;*)
		bMsg1143 : BOOL; (*Voltage negative sequence*) (*OldName:newPV; Cycle:5;*)
		bMsg1144 : BOOL; (*Current negative sequence*) (*OldName:newPV; Cycle:5;*)
		bMsg1175 : BOOL; (*mains failure*) (*OldName:AMM_W11xx[]; Cycle:5;*)
		bMsg1189 : BOOL; (*release from synchronization missing*) (*OldName:AMM_W11xx[]; Cycle:5;*)
		bMsg1209 : BOOL; (*mains circuit breaker position signal failure*) (*OldName:AMM_W12xx[]; Cycle:5;*)
		bMsg1210 : BOOL; (*mains circuit breaker opening failure*) (*OldName:AMM_W12xx[]; Cycle:5;*)
		bMsg1211 : BOOL; (*mains circuit breaker closing failure*) (*OldName:AMM_W12xx[]; Cycle:5;*)
		bMsg1212 : BOOL; (*mains circuit breaker o-signal failure*) (*OldName:AMM_W12xx[]; Cycle:5;*)
		bMsg1213 : BOOL; (*mains circuit breaker 1-signal failure*) (*OldName:AMM_W12xx[]; Cycle:5;*)
		bMsg1214 : BOOL; (*mains circuit breaker overload/short circuit*) (*OldName:AMM_W12xx[]; Cycle:5;*)
		bMsg1216 : BOOL; (*bus bar voltage sensor failure*) (*OldName:AMM_W12xx[]; Cycle:5;*)
		bMsg1217 : BOOL; (*generator circuit breaker position signal failure*) (*OldName:AMM_W12xx[]; Cycle:5;*)
		bMsg1218 : BOOL; (*generator circuit breaker opening failure*) (*OldName:AMM_W12xx[]; Cycle:5;*)
		bMsg1219 : BOOL; (*generator circuit breaker closing failure*) (*OldName:AMM_W12xx[]; Cycle:5;*)
		bMsg1220 : BOOL; (*generator circuit breaker o-signal failure*) (*OldName:AMM_W12xx[]; Cycle:5;*)
		bMsg1221 : BOOL; (*generator circuit breaker 1-signal failure*) (*OldName:AMM_W12xx[]; Cycle:5;*)
		bMsg1222 : BOOL; (*generator manual circuit breaker open*) (*OldName:AMM_W12xx[]; Cycle:5;*)
		bMsg1235 : BOOL; (*generator circuit breaker closed*) (*OldName:AMM_B12xx[]; Cycle:5;*)
		bMsg1236 : BOOL; (*generator circuit breaker opened*) (*OldName:AMM_B12xx[]; Cycle:5;*)
		bMsg2139 : BOOL; (*synchronizing running*) (*OldName:AMM_B21xx[]; Cycle:5;*)
		bMsg2330 : BOOL; (*mid voltage CB failure*)
		bMsg2354 : BOOL; (*earth fault bus bar*)
		bMsg2366 : BOOL; (*generator circuit breaker closing failure*)
		bMsg2688 : BOOL; (*Generator current at synchronization too high*) (*OldName:newPv;Cycle:5*)
		bMsg2692 : BOOL; (*generator circuit breaker opening failure*) (*OldName:newPV; Cycle:5;*)
		bMsg2693 : BOOL; (*generator circuit breaker opening failure*) (*OldName:newPV; Cycle:5;*)
		bMsg2730 : BOOL; (*low voltage CB failure*) (*OldName:AMM_W33xx[]; Cycle:5;*)
		bMsg2801 : BOOL; (*module blocked by grid connection conditions*) (*OldName:NewbMsg; Cycle:5;*)
		bMsg2901 : BOOL; (*synchronization selection OFF*) (*OldName:NewPv; Cycle:5;*)
		bMsg2902 : BOOL; (*synchronization selection MAN*) (*OldName:NewPv; Cycle:5;*)
		bMsg2903 : BOOL; (*synchronization selection AUT*) (*OldName:NewPv; Cycle:5;*)
		bMsg2934 : BOOL; (*module blocked by grid connection conditions after mains failure*) (*OldName:NewPv; Cycle:5;*)
		bMsg3253 : BOOL; (*begin maintenance/testbench mode*) (*OldName:AMM_B32xx[]; Cycle:5;*)
		bMsg3254 : BOOL; (*end   maintenance/testbench mode*) (*OldName:AMM_B32xx[]; Cycle:5;*)
		bMsg3263 : BOOL; (*mains circuit breaker closed*) (*OldName:AMM_B32xx[]; Cycle:5;*)
		bMsg3264 : BOOL; (*mains circuit breaker opened*) (*OldName:AMM_B32xx[]; Cycle:5;*)
		bMsg3265 : BOOL; (*demand close GCB*) (*OldName:AMM_B32xx[]; Cycle:5;*)
		bMsg3266 : BOOL; (*mains failure on*) (*OldName:AMM_B32xx[]; Cycle:5;*)
		bMsg3267 : BOOL; (*mains failure off*) (*OldName:AMM_B32xx[]; Cycle:5;*)
		bMsg3269 : BOOL; (*generator de-energized*)
		bMsg3296 : BOOL; (*demand generator excitation off*)
		bMsg3297 : BOOL; (*demand generator excitation on*)
		bMsg3329 : BOOL; (*earth circuit breaker closed, france country specific*) (*OldName:AMM_W33xx[]; Cycle:5;*)
		bMsg3352 : BOOL; (*disconnecting circuit breaker opened, france country specific*) (*OldName:AMM_W33xx[]; Cycle:5;*)
		bMsg3400 : BOOL; (*module blocked by no operating release from sy or cooling water temp.low*) (*OldName:NewPv; Cycle:5;*)
		bMsg3412 : BOOL; (*mains monitoring device failure*) (*OldName:AMM_W34xx[]; Cycle:5;*)
		bMsg3575 : BOOL; (*mains failure GTE2666, france country specific*) (*OldName:AMM_W35xx[]; Cycle:5;*)
		bMsg3576 : BOOL; (*mains failure TGS, france country specific*) (*OldName:AMM_W35xx[]; Cycle:5;*)
		bMsg3577 : BOOL; (*mains failure C13.100, france country specific*) (*OldName:AMM_W35xx[]; Cycle:5;*)
		bMsg9244 : BOOL; (*generator circuit breaker not ready*)
		bMsg9245 : BOOL; (*generator circuit breaker not racked-in*)
		bMsg9304 : BOOL; (*generator circuit breaker closing time deviation high*)
		bMsg9331 : BOOL; (*maintenance request generator circuit breaker*)
		tiGCB_ClosTime : TIME; (*generator circuit breaker closing time*)
		tiGCB_ClosTimeOld : TIME; (*generator circuit breaker closing time old*)
		bMsg1041Set : BOOL; (*power signal missing*)
		bMsg1042Set : BOOL; (*power signal overload*)
		bMsg2801Set : BOOL; (*module blocked by grid connection conditions*)
		bMsg2934Set : BOOL; (*module blocked by grid connection conditions after mains failure*)
		bDemGenExcOff : BOOL; (*demand generator excitation off*)
		bGenExcOff : BOOL; (*generator excitation off*)
		bMsg9083 : BOOL; (*LCB open*)
		bMsg9084 : BOOL; (*LCB closed*)
		tGCB : ARRAY[0..2]OF GCB2VIS_Struct; (* LV GCB *)
		bMsg9085 : BOOL; (*Parameters saved to the GCB*)
		bMsg9382 : BOOL; (*GCB contact wear over 80%*)
		bMsg9383 : BOOL; (*GCB contact wear over 95%*)
	END_STRUCT;
END_TYPE

(*END_MM2VIS*)

TYPE
	VIS2MM_Struct : 	STRUCT
		bGCB_MOf : BOOL; (*gcb manual off command button*) (*OldName:DI_GCB_MOF; Cycle:5;*)
		bGCB_MOn : BOOL; (*gcb manual on  command button*) (*OldName:DI_GCB_MON; Cycle:5;*)
		bMCB_MOf : BOOL; (*mcb manual off command button*) (*OldName:DI_MCB_MOF; Cycle:5;*)
		bMCB_MOn : BOOL; (*mcb manual on  command button*) (*OldName:DI_MCB_MON; Cycle:5;*)
		iIdx_SyOMSS : DINT; (*synchronization operating mode selection*) (*OldName:newPv; Cycle:5;*)
		bServiceBegin : BOOL; (*service begin (VIS button)*) (*OldName:bServiceBegin; Cycle:5;*)
		iGCB_OnCnt : DINT; (*generator circuit breaker cycle counter*)
		iModule : INT; (*HMI/SYS/Module/Module number setted*)
		tGCB : ARRAY[0..2]OF VIS2GCB_Struct; (* LV GCB *)
	END_STRUCT;
	cb_Struct : 	STRUCT
		enable : BOOL;
		rdy : BOOL;
		racked_in : BOOL;
		opf : BOOL;
		on : BOOL;
		off : BOOL;
		dmnd_sy : BOOL;
		remote : BOOL;
		man_off : BOOL;
		man_on : BOOL;
		release : BOOL;
		aut_on2dead_bb : BOOL;
		man_on2dead_bb : BOOL;
		eng_demanded : BOOL;
		eng_run : BOOL;
		eng_oper : BOOL;
		esl : BOOL;
		edc_in : BOOL;
		edc : BOOL;
		all_other_gcb_off : BOOL;
		other_gcb_on : BOOL;
		other_gen_parallel : BOOL;
		rel_sy_puls : BOOL;
		rel_island : BOOL;
		dmnd_on : BOOL;
		dmnd_off : BOOL;
		command_on : BOOL;
		command_off : BOOL;
		rel_trip : BOOL;
		mon_release : BOOL;
		mdl : BOOL;
		mrc : BOOL;
		alarm : BOOL;
		alm_psf : BOOL;
		alm_opf : BOOL;
		alm_cf : BOOL;
		alm_0sf : BOOL;
		alm_1sf : BOOL;
		alm_ol : BOOL;
	END_STRUCT;
	mns_Struct : 	STRUCT
		enable : BOOL;
		ok : BOOL;
		return_rest_time : DINT;
	END_STRUCT;
	Perm_SY_Struct : 	STRUCT
		iIdx_SyOMSS : DINT; (*synchronization operating mode selection*)
		iGCB_OnCnt : DINT; (*generator circuit breaker cycle counter*)
		rTB_PermValue02 : REAL; (*spare permanent value for testbench- replace with new vars of same lenght, when needed*) (*OldName:new PV;Cycle:2;*)
		rTB_PermValue03 : REAL; (*spare permanent value for testbench- replace with new vars of same lenght, when needed*) (*OldName:new PV;Cycle:2;*)
		rTB_PermValue04 : REAL; (*spare permanent value for testbench- replace with new vars of same lenght, when needed*) (*OldName:new PV;Cycle:2;*)
		rTB_PermValue05 : REAL; (*spare permanent value for testbench- replace with new vars of same lenght, when needed*) (*OldName:new PV;Cycle:2;*)
		rTB_PermValue06 : REAL; (*spare permanent value for testbench- replace with new vars of same lenght, when needed*) (*OldName:new PV;Cycle:2;*)
		rTB_PermValue07 : REAL; (*spare permanent value for testbench- replace with new vars of same lenght, when needed*) (*OldName:new PV;Cycle:2;*)
		rTB_PermValue08 : REAL; (*spare permanent value for testbench- replace with new vars of same lenght, when needed*) (*OldName:new PV;Cycle:2;*)
		rTB_PermValue09 : REAL; (*spare permanent value for testbench- replace with new vars of same lenght, when needed*) (*OldName:new PV;Cycle:2;*)
		rTB_PermValue10 : REAL; (*spare permanent value for testbench- replace with new vars of same lenght, when needed*) (*OldName:new PV;Cycle:2;*)
	END_STRUCT;
	OpMode_Switches : 	STRUCT
		iIdx_OMS_Hw : INT; (* index of hardware operation mode selector switch *)
		iIdx_RMS_Hw : INT; (* index of hardware request mode selector switch *)
		iIdx_SyOMS_Hw : INT; (* index of hardware synchronisation operation mode selector switch *)
		bGoodQual : BOOL; (* Global GoodQual Bit for all 3 hw-switches *)
	END_STRUCT;
	GCB2VIS_Struct : 	STRUCT
		bEna : BOOL; (* X20CS1030_xxx_xx_GCB was found*)
		rSave : REAL; (* Save process*)
		rLoad : REAL; (* Load process*)
		iState : UINT; (* Current State of Statemachine*)
		iError : UINT; (* Error numbers from Modbus*)
		iType : INT; (* Types: 1 = ABB EMax, 2 = Schneider MTZ *)
		iNumOp : DINT; (* Number of GCB operations *)
		iNumPT : DINT; (* Number of GCB protection trips *)
		bClosed : BOOL; (* TRUE = GCB is closed *)
		bFail : BOOL; (* TRUE = GCB failure *)
		bRacked : BOOL; (* TRUE = GCB is racked in *)
		rU_Nom : REAL; (* [V] Nominal Voltage *)
		rI_Nom : REAL; (* [A] Nominal Current *)
		rU_Act : REAL; (* [V] Actual Voltage *)
		rI_Act_L1 : REAL; (* [A] Actual Current L1 *)
		rI_Act_L2 : REAL; (* [A] Actual Current L2 *)
		rI_Act_L3 : REAL; (* [A] Actual Current L3 *)
		rWear : REAL; (* [0-1] contact wear of GCB *)
	END_STRUCT;
	VIS2GCB_Struct : 	STRUCT
		bLoad : BOOL; (* TRUE = Load parameters from GCB *)
		bSave : BOOL; (* TRUE = Save parameters to GCB *)
		bCalc : BOOL; (* TRUE = Calc parameters from I_Nom *)
		rI_GenNom : REAL; (* [A] Nominal Generator Current *)
		rt1 : REAL; (* [s] Short circuit protection delay t1 / tr *)
		rt2 : REAL; (* [s] Overload protection delay t2 / tsd *)
		rI1 : REAL; (* [A] Overload protection current I1 / Ir *)
		rI2 : REAL; (* [A] Short circuit protection delayed current I2 / Isd *)
		rI3 : REAL; (* [A] short circuit protection instantaneous I3 / Ii *)
	END_STRUCT;
END_TYPE
```

### module_SYPara.typ
```iecst
TYPE
	PROGRAMMER_INFO : 	STRUCT
		DO_NOT_SORT_PARA : STRING[40] := 'DO NOT CHANGE PARAMETER SORTING!'; (*DO NOT CHANGE PARAMETER SORTING!*) (*ADD NEW PARAMETER ONLY AT THE END OF THE Para STRUCTURE. DO NOT DELETE existing Para items.*)
	END_STRUCT;
	Para_SY_struct : 	STRUCT
		rN_EngNom : REAL; (*PARA [12128]: engine nominal speed [1/min]*) (*OldName:n_nenn; Cycle:5;*)
		rU_Gen_Nom : ARRAY[0..2]OF REAL; (*PARA [11597], [11598]: generator nominal voltage [V]*) (*OldName:usUNennGen[1]; Cycle:5;*)
		bGlowIgnPrevActive : BOOL; (*PARA [12089]: glow ignition prevention active *) (*OldName:sel_GlowIgnPrevent; Cycle:5;*)
		bRemoteReqActive : BOOL; (*PARA [12091]: remote request active *) (*OldName:bRemoteReqAct; Cycle:5;*)
		rP_LimLo : REAL; (*PARA [12208]: power signal missing limit low  *) (*OldName:Z_GW_LSA; Cycle:5;*)
		rP_HyLo : REAL; (*PARA [12206]: power signal missing limit hysteresis low  *) (*OldName:HY_LSA; Cycle:5;*)
		rP_LimHi : REAL; (*PARA [12207]: power signal overload limit high  *) (*OldName:GW_LSU; Cycle:5;*)
		rP_HyHi : REAL; (*PARA [12205]: power signal overload limit hysteresis high  *) (*OldName:HY_LSU; Cycle:5;*)
		tiMainsOkDelay : TIME; (*PARA [12216]: mains return delay *) (*OldName:PT_MNS_OK; Cycle:5;*)
		rP_LS_LimHi : REAL; (*PARA [12212]: generator power limit high (load shedding)(% Pnom) *) (*OldName:GW_P_MAX; Cycle:5;*)
		rP_LS_HyHi : REAL; (*PARA [12209]: generator power hysteresis limit high (load shedding)(% Pnom) *) (*OldName:HY_P_MAX; Cycle:5;*)
		tiP_LS_LimHi : TIME; (*PARA [12219]: generator power limit high delay (load shedding)(% Pnom) *) (*OldName:TW_P_MAX; Cycle:5;*)
		rP_LS_LimLo : REAL; (*PARA [12213]: generator power limit low warning (load shedding)(% Pnom) *) (*OldName:GW_P_MIN_W; Cycle:5;*)
		rP_LS_HyLo : REAL; (*PARA [12210]: generator power hysteresis limit low warning (load shedding)(% Pnom) *) (*OldName:newPv; Cycle:5;*)
		tiP_LS_LimLo : TIME; (*PARA [12220]: generator power limit low warning delay (load shedding)(% Pnom) *) (*OldName:TW_P_MIN_W; Cycle:5;*)
		rP_LS_LimLoLo : REAL; (*PARA [12214]: generator power limit low shutdown (load shedding)(% Pnom) *) (*OldName:GW_P_MIN_A; Cycle:5;*)
		rP_LS_HyLoLo : REAL; (*PARA [12211]: generator power hysteresis limit low shutdown (load shedding)(% Pnom) *) (*OldName:HY_P_MIN; Cycle:5;*)
		tiP_LS_LimLoLo : TIME; (*PARA [12221]: generator power limit low shutdown delay (load shedding) *) (*OldName:TW_P_MIN_A; Cycle:5;*)
		rN_LS_LimLo : REAL; (*PARA [12204]: engine speed limit low (load shedding) [1/min]*) (*OldName:GW_DR_MIN; Cycle:5;*)
		rN_LS_HyLo : REAL; (*PARA [12203]: engine speed hysteresis limit low (load shedding) [1/min]*) (*OldName:HY_DR_MIN; Cycle:5;*)
		tiN_LS_LimLo : TIME; (*PARA [12218]: engine speed limit low delay (load shedding) [1/min]*) (*OldName:TW_DR_MIN; Cycle:5;*)
		iEng_Motortype : INT; (* Para engine motortype *) (*OldName:motortyp; Cycle:5;*)
		iCountry : INT; (*PARA [12196]: code for country specific functions *) (*OldName:newPv; Cycle:5;*)
		bMCB_SyMMD2 : BOOL; (*PARA [12189]: synchronization mcb with MMUsynch 2 *) (*OldName:bMMU2syMCB; Cycle:5;*)
		bSyActive : BOOL; (*PARA [12195]: synchronization functions active *) (*OldName:bSynch; Cycle:5;*)
		bMSy : BOOL; (*PARA [12193]: connected to master sy/interlock panel *) (*OldName:msy; Cycle:5;*)
		bMCB_Enable : BOOL; (*PARA [12187]: mains circuit breaker enable (mcb controlled by esy) *) (*OldName:mcb[1].enable; Cycle:5;*)
		bC_CB_Enable : BOOL; (*PARA [12181]: customer circuit breaker (gcb0 = custom generator/engine) enable *) (*OldName:gcb[0].enable; Cycle:5;*)
		bMns_Enable : BOOL; (*PARA [12191]: mains monitoring enable *) (*OldName:mains[1].enable; Cycle:5;*)
		bOnlyIsland_Enable : BOOL; (*PARA [12194]: only island operation (without MSY) enable *) (*OldName:sel_only_island; Cycle:5;*)
		bIslandOp_Enable : BOOL; (*PARA [12184]: island operation (without MSY) enable *) (*OldName:sel_island; Cycle:5;*)
		bBS_Enable : BOOL; (*PARA [12179]: black start enable *) (*OldName:sel_black_start; Cycle:5;*)
		bBS_Acc_Active : BOOL; (*PARA [12178]: black start accelerated active *) (*OldName:sel_black_start_15s; Cycle:5;*)
		rN_BS_Acc_LimHi : REAL; (*PARA [12202]: black start accelerated speed limit high (for engine operation)[rpm] *) (*OldName:bs_15s_rpm_lim_hi; Cycle:5;*)
		bBS_OnlyMan : BOOL; (*PARA [12180]: black start only manual enable *) (*OldName:sel_only_man_black; Cycle:5;*)
		bADL_Enable : BOOL; (*PARA [12177]: anti detonation logic enable *) (*OldName:sel_anti_detonat_logic; Cycle:5;*)
		bMIF_Enable : BOOL; (*PARA [12190]: micro interruption filter enable *) (*OldName:sel_mi_filter_activ; Cycle:5;*)
		bEngOpAfterMIF_Enable : BOOL; (*PARA [12182]: engine operation after micro interruption filter enable *) (*OldName:sel_op_after_MIF; Cycle:5;*)
		bMCB_ReSw2Mns_Enable : BOOL; (*PARA [12188]: mains circuit breaker reswitch to mains enable *) (*OldName:sel_reswitch_to_mains; Cycle:5;*)
		bGenDeexit_Enable : BOOL; (*PARA [12183]: generator deexitation enable *) (*OldName:sel_de_excit; Cycle:5;*)
		bMCB_Ctr_Cust : BOOL; (*PARA [12186]: mains circuit breaker controlled by customer *) (*OldName:sel_mcb_ctrl_c; Cycle:5;*)
		tiMIF : TIME; (*PARA [12217]: micro interruption filter delay time *) (*OldName:PT_MIF; Cycle:5;*)
		rN_EngStart_LimHi : REAL; (*PARA [11296]: speed engine start limit high [1/min]*) (*OldName:GW_DREHZ; Cycle:5;*)
		rN_EngStart_HyHi : REAL; (*PARA [11295]: speed engine start limit high hysteresis [1/min]*) (*OldName:HY_DREHZ; Cycle:5;*)
		rU_Gen_DeEx_LimLo : REAL; (*PARA [12215]: generator voltage deexcitation limit low*) (*OldName:GW_GEN_OSP; Cycle:5;*)
		bGridCode_Active : BOOL; (*PARA [11055]: Gride Code active*) (*OldName:bGridCode; Cycle:5;*)
		bLoadShedPara_Visible : BOOL; (*PARA [12185]: isolated operation/limits load shedding visible*) (*OldName:bIsolOperation; Cycle:5;*)
		iMnsPath_Visible : INT; (*PARA [12199]: connection mains circuit breaker visible*) (*OldName:usVisuNetPath; Cycle:5;*)
		bMnsOk_Visible : BOOL; (*PARA [12192]: symbol mains ok status without mains path visible*) (*OldName:bVisuNetOK; Cycle:5;*)
		iGenPathDown_Visible : INT; (*PARA [12197]: symbol down generator cb - path visible(0=no symbol, 1=transformer, 2=circuit breaker)*) (*OldName:usVisuGenPathDown; Cycle:5;*)
		iGenPathUp_Visible : INT; (*PARA [12198]: symbol up generator cb - path visible(0=no symbol, 1=transformer, 2=circuit breaker)*) (*OldName:usVisuGenPathUp; Cycle:5;*)
		iMnsPathDown_Visible : INT; (*PARA [12200]: symbol down mains cb - path visible(0=no symbol, 1=transformer, 2=circuit breaker)*) (*OldName:usVisuNetPathDown; Cycle:5;*)
		iMnsPathUp_Visible : INT; (*PARA [12201]: symbol up mains cb - path visible(0=no symbol, 1=transformer, 2=circuit breaker)*) (*OldName:usVisuNetPathUp; Cycle:5;*)
		bP_LoadReject_Active : BOOL; (*PARA [12890]: Load rejection funcitons active *) (*OldName:newPv; Cycle:5;*)
		bBB_ClosCondLimits_Active : BOOL; (*PARA [13172]: Busbar closing condition limit active *) (*OldName:newPv; Cycle:5;*)
		rU_BB_ClosCond_LimLo_Norm : REAL; (*PARA [13173]: Busbar closing condition norm voltage lower limit *) (*OldName:newPv; Cycle:5;*)
		rU_BB_ClosCond_LimHi_Norm : REAL; (*PARA [13174]: Busbar closing condition norm voltage higher limit *) (*OldName:newPv; Cycle:5;*)
		rU_BB_ClosCond_Hy_Norm : REAL; (*PARA [13175]: Busbar closing condition norm voltage hysteresis *) (*OldName:newPv; Cycle:5;*)
		rF_BB_ClosCond_LimLo : REAL; (*PARA [13176]: Busbar closing condition frequency lower limit *) (*OldName:newPv; Cycle:5;*)
		rF_BB_ClosCond_LimHi : REAL; (*PARA [13177]: Busbar closing condition frequency higher limit *) (*OldName:newPv; Cycle:5;*)
		rF_BB_ClosCond_Hy : REAL; (*PARA [13178]: Busbar closing condition frequency hysteresis *) (*OldName:newPv; Cycle:5;*)
		tiBB_ClosCond_Delay : TIME; (*PARA [13179]: Busbar closing condition delay time *) (*OldName:newPv; Cycle:5;*)
		tiBB_ClosCondAftMnsFail_Delay : TIME; (*PARA [13180]: Busbar closing condition delay time after mains failure *) (*OldName:newPv; Cycle:5;*)
		tiMCB_COf_GCB_OpF : TIME; (*PARA [13309]: delay time opening MCB in case of GCB opening failure*) (*OldName:newPv; Cycle:5;*)
		rP_Red_TempMax_GenCB_Rate : REAL; (*PARA [13272]: Setpoint power reduction temp. max generator switch gear*) (*OldName:newPv; Cycle:5;*)
		bP_Red_TempMax_GenCB_Active : BOOL; (*PARA [13271]: activation power reduction temp. max generator switch gear*) (*OldName:newPv; Cycle:5;*)
		rI_GenNom : ARRAY[0..2]OF REAL; (*PARA [11750], [11751]: nominal current generator [0..65kA] *) (* OldName:usINennGen; Cycle: 5*)
		bGCB_MainsCutOff_Active : BOOL; (*PARA [13263]: mains cut off with generator circuit breaker active*) (*OldName:sel_gcb_mains_cut_off_Enable; Cycle:5;*)
		rU_BusNom : ARRAY[0..2]OF REAL; (*PARA [11851], [11852]: nominal voltage bus [70V..65kV] *) (* OldName:usUNennBus; Cycle: 5*)
		bRej2houseload : BOOL; (*PARA [14079]: Fangen im Eigenbedarf aktiv?*)
		bBB_AfMnsF_ClosCondLimits_Active : BOOL; (*PARA [14136]: Busbar closing condition limit after mains failure active *) (*OldName:newPv; Cycle:5;*)
		rU_BB_AfMnsF_ClosCond_LimLo_Norm : REAL; (*PARA [14137]: Busbar closing condition norm voltage lower limit after mains failure*) (*OldName:newPv; Cycle:5;*)
		rU_BB_AfMnsF_ClosCond_LimHi_Norm : REAL; (*PARA [14138]: Busbar closing condition norm voltage higher limit after mains failure*) (*OldName:newPv; Cycle:5;*)
		rU_BB_AfMnsF_ClosCond_Hy_Norm : REAL; (*PARA [14139]: Busbar closing condition norm voltage hysteresis after mains failure*) (*OldName:newPv; Cycle:5;*)
		rF_BB_AfMnsF_ClosCond_LimLo : REAL; (*PARA [14140]: Busbar closing condition frequency lower limit after mains failure*) (*OldName:newPv; Cycle:5;*)
		rF_BB_AfMnsF_ClosCond_LimHi : REAL; (*PARA [14141]: Busbar closing condition frequency higher limit after mains failure*) (*OldName:newPv; Cycle:5;*)
		rF_BB_AfMnsF_ClosCond_Hy : REAL; (*PARA [14142]: Busbar closing condition frequency hysteresis after mains failure*) (*OldName:newPv; Cycle:5;*)
  		bMMDSynch_Act : ARRAY[0..2]OF BOOL; (*PARA [11714], [11715]: synchronization of MMDsynch active *) (* OldName:bMMUSynchAct; Cycle: *)
  		rTi_SynchImpMin : ARRAY[0..2]OF REAL; (*PARA [11837], [11838]: minimum impulse width of DO4 [0,04..0,5s] *) (* OldName:usImpDO4Min; Cycle: *)
  		rTi_SynchSwitchDel : ARRAY[0..2]OF REAL; (*PARA [11839], [11840]: witching delay of the relay switched with DO4 [40..300ms] *) (* OldName:usSwitchDelDO4; Cycle: *)
		iGCB_OnCnt_LimHi : DINT; (*PARA [14495]: generator circuit breaker switching cycles maintenance request*)
		rP_LimHiHi : REAL; (*PARA [12559]: power signal overload  isolated mode *) (*OldName; Cycle:5;*)
		ti_P_LimHiHi : TIME; (* PARA [14510]: power signal overload  isolated mode delay *) (*OldName; Cycle:5;*)
		iSel_Customer : DINT; (*PARA [14950]: 0 = no special, 1 = AB Energy, 2 = Aggreko, 3 = 2G, etc.... *)
	END_STRUCT;
END_TYPE
```

### module_SY.var
```iecst
VAR
	IN_SY : IN_SY_struct;
	OUT_SY : OUT_SY_struct;
	MM2VIS : MM2VIS_Struct;
	VIS2MM : VIS2MM_Struct;
	Para : Para_SY_struct;
	ParaFactoryDefault : Para_SY_struct;
	pm : Para_SY_struct;
	xEngType : EngType; (*engine type*)
	xOpMode : OpMode; (*engine operation mode*)
	gcb : cb_Struct; (*generator circuit breaker*)
	ccb : cb_Struct; (*customer circuit breaker(generator)*)
	mcb : cb_Struct; (*mains circuit breaker*)
	mains : mns_Struct; (*mains*)
	bOMSS_Stop : BOOL; (*engine operation mode selection*)
	bOMSS_Man : BOOL; (*engine operation mode selection*)
	bOMSS_Aut : BOOL; (*engine operation mode selection*)
	bOMSS_Test : BOOL; (*engine operation mode selection*)
	bOMSS_Scav : BOOL; (*engine operation mode selection*)
	bOMSS_MAT : BOOL; (*engine operation mode selection*)
	bSyOMSS_Off : BOOL; (*synchronization operating mode selection OFF*)
	bSyOMSS_Man : BOOL; (*synchronization operating mode selection MANUAL*)
	bSyOMSS_Aut : BOOL; (*synchronization operating mode selection AUTO*)
	bMCB_GnlWarning : BOOL; (*Vis mains circuit breaker general warning*)
	bGCB_GnlWarning : BOOL; (*Vis generator circuit breaker general warning*)
	ANW_ENTR : BOOL;
	bb_alive : BOOL; (*bus bar alive*)
	bb_dead : BOOL; (*bus bar dead*)
	bGnlTrip : BOOL;
	bGnlTrip1 : BOOL;
	bGnlTrip2 : BOOL;
	bGnlTrip3 : BOOL;
	bGnlWarning : BOOL;
	bMainsReturn : BOOL; (*mains ok with delay*)
	BLOCK_NS : BOOL; (*demand lock customer mcb while running island operation*)
	BLOUT : BOOL; (*demand blackout for demand load shedding*)
	bMsg1041_Test : BOOL; (*test*)
	bMsg1042_Test : BOOL; (*test*)
	dmnd_black_start : BOOL; (*demand bloack-out start for demand load shedding*)
	bDem_Island : BOOL; (*Demand island*)
	DR_MIN : BOOL; (*Speed below 1400 rpm*)
	gcb_opf_delay : BOOL; (*opening mcb after delay *)
	GEN_OSP : BOOL; (*Feedback Generator without voltage*)
	bN_EngStart : BOOL; (*engine start speed*)
	P_MAX : BOOL; (*Power above > 95%*)
	bRelease_Island : BOOL; (*release island for W1175 and block engine*)
	rel_load_shedd : BOOL; (*load shedding ok*)
	ton_gcb_dmnd_sy : TON; (*gcb demand synchronization*)
	any_gcb_on_bb : BOOL; (*any gcb on bus bar*)
	other_gcb_on : BOOL; (*other gcb on*)
	other_gcb_off : BOOL; (*other gcb off*)
	all_gcb_off_bb : BOOL; (*all gcb off bus bar*)
	any_eng_oper_and_gcb_on_bb : BOOL; (*any engine operating an gcb on bus bar*)
	no_eng_run_bb : BOOL; (*no engine runing bus bar*)
	any_eng_run_bb : BOOL; (*any engine runing bus bar*)
	any_gcb_psf_bb : BOOL; (*any gcb position signal failure bus bar*)
	any_gcb_opf_bb : BOOL; (*any gcb opening failure bus bar*)
	any_gcb_alarm_bb : BOOL; (*any gcb alarm bus bar*)
	any_gcb_edc_bb : BOOL; (*any gcb demand close to dead bus bar *)
	rel_gcb_on2d_bb : BOOL; (*release gcb on to dead bus bar*)
	rel_mcb_on2d_bb : BOOL; (*release mcb on to dead bus bar*)
	bP_Lo : BOOL; (*power low - open gcb, power signal missing*)
	rel_sy_puls : BOOL; (* release synchronizing pulse *)
	pulse_sy_line : BOOL; (*pulse synch line*)
	rU_Gen_Norm : REAL; (*generator voltage [%]*)
	dmnd_synchline : BOOL; (*demand_synchline*)
	mcb_man_on2dead_bb : BOOL; (*mcb manual closing to dead bus bar*)
	mcb_aut_on2dead_bb : BOOL; (*mcb autom. closing to dead bus bar*)
	rel_i_adl : BOOL; (*release island operation from anti detonation logic*)
	sel_gcb_mains_cut_off : BOOL; (*select cut off from mains with gcb when mains failure*)
	rel_black_start : BOOL; (*release black start*)
	bGen_DeExc_Rdy : BOOL; (*generator deexitation ready*)
	bGen_DeExc_Err : BOOL; (*generator deexitation failed*)
	P_MIN_W : BOOL; (*generator power low for load shedding warning*)
	P_MIN_A : BOOL; (*generator power low for load shedding trip*)
	bGCB_MOn : BOOL; (*generator cb manual on command form visu button*)
	bGCB_MOf : BOOL; (*generator cb manual on command form visu button*)
	bMCB_MOn : BOOL; (*mains cb manual on command form visu button*)
	bMCB_MOf : BOOL; (*mains cb manual on command form visu button*)
	bTestBenchMode : BOOL; (*test bench mode active*)
	iEngNr : INT; (*engine number according IP address*)
	bAMM_ClosCond_Ok : BOOL; (* Closing condition result*)
	bBBClosCond_Fault : BOOL; (* Closing conditions fault detected - status after mains failure*)
	bAMM_AfMnsF_ClosCond_Ok : BOOL; (* Closing condition result*)
	bGCBctd : BOOL; (*gcb closing time deviation*)
	bResetWarning : BOOL; (*reset from AmmBase*)
	bGenDeexitDem : BOOL; (*demand generator deexcitation*)
	bB9085_GCB_ParaSaved : BOOL; (* B9085 Parameters saved to the GCB *)
	bW9382_GCB_Wear80 : BOOL; (* W9382 GCB contact wear over 80% *)
	bW9383_GCB_Wear95 : BOOL; (* W9383 GCB contact wear over 95% *)
END_VAR
VAR CONSTANT
	iPakistan : INT := 92; (*country code*)
	iHolland : INT := 31; (*country code*)
END_VAR
VAR
	bNoInitDetected : BOOL := FALSE; (*allways true, except 1cycle on init up*)
	bF_BB_ClosCond : BOOL := 0;
	bF_BB_AfMnsF_ClosCond : BOOL := 0;
END_VAR
```

### Program Logical/Synchronization/default_SY (IEC, version 4.10.0) - values

#### default_SYCyclic.st
```iecst
(*******************************************************************************
default		values

This code is confidential and proprietary to the INNIO Company.
It may not be used in any form, or reproduced in any manner,
without the express written permission of the INNIO Company.
Copyright, INNIO Company, 2019

Customized modifications: -
------------------------

History:
-------
V0.00.0	24.04.2012	lettenb.	new
V3.90.0	27.11.2012	lettenb.	corr.for P3 startup
V3.99.0	25.02.2012	lettenb.	3329,3352,3575,3576,3577 added (integration V3.30-V3.40)
V4.00.0 11.06.2014	lettenb.	tOnly_Island, tEngDemIsland added
		18.06.2014				tBB_Alive.Di removed, bugfix
V4.03.0	22.07.2015				2692,2693,2801 new, dyn.gridcode III(thaler)
		14.08.2015				IN_SY.tOnly_Island.Di init removed (see TBMode: OUT_SY.bOnly_Island	logic FOR standard mode corr. removed) (bugfix/pfanzagl)
V4.05.0	03.01.2018	lettenb.	tMnsOk_AfMnsF_ClosCond_Ok added, grid code logic(thaler)
V4.07.0	31.10.2018	lettenb.	tMidVoltCB_Failure added
V4.10.0	23.11.2020	lettenb.	tGndFault_BB added

Instructions for use:
--------------------
Outstandings:
------------
*******************************************************************************)
PROGRAM _CYCLIC

	(* default TRUE setting for not existing Di's *)
	(* note: existing but not used Di's if necessary have to be setted to TRUE by hardware *)
	IN_SY.tGCB_Rac.Di			:=	IN_SY.tGCB_Rac.Di			OR	NOT IN_SY.tGCB_Rac.GoodQual;
	IN_SY.tGCB_Rdy.Di			:=	IN_SY.tGCB_Rdy.Di			OR	NOT IN_SY.tGCB_Rdy.GoodQual;
	IN_SY.tGCB_MRC.Di			:=	IN_SY.tGCB_MRC.Di			OR	NOT IN_SY.tGCB_MRC.GoodQual;
	IN_SY.tGCB_AGO.Di			:=	IN_SY.tGCB_AGO.Di			OR	NOT IN_SY.tGCB_AGO.GoodQual;
	IN_SY.tGCB_RI.Di			:=	IN_SY.tGCB_RI.Di			OR	NOT IN_SY.tGCB_RI.GoodQual;

	IN_SY.tRel_I.Di				:=	IN_SY.tRel_I.Di				OR	NOT IN_SY.tRel_I.GoodQual;
	IN_SY.tRel_BS.Di			:=	IN_SY.tRel_BS.Di			OR	NOT IN_SY.tRel_BS.GoodQual;
	IN_SY.tRel_LS.Di			:=	IN_SY.tRel_LS.Di			OR	NOT IN_SY.tRel_LS.GoodQual;

	IN_SY.tMCB_Rac.Di			:=	IN_SY.tMCB_Rac.Di			OR	NOT IN_SY.tMCB_Rac.GoodQual;
	IN_SY.tMCB_Rdy.Di			:=	IN_SY.tMCB_Rdy.Di			OR	NOT IN_SY.tMCB_Rdy.GoodQual;
	IN_SY.tMCB_OL.Di			:=	IN_SY.tMCB_OL.Di			OR	NOT IN_SY.tMCB_OL.GoodQual;
	IN_SY.tMCB_Rem.Di			:=	IN_SY.tMCB_Rem.Di			OR	NOT IN_SY.tMCB_Rem.GoodQual;

	IN_SY.tMnsOk.Di				:=	IN_SY.tMnsOk.Di				OR	NOT IN_SY.tMnsOk.GoodQual;
	IN_SY.tMns_MDF.Di			:=	IN_SY.tMns_MDF.Di			OR	NOT IN_SY.tMns_MDF.GoodQual;

	IN_SY.tC_CB_Off.Di			:=	IN_SY.tC_CB_Off.Di			OR	NOT IN_SY.tC_CB_Off.GoodQual;
	IN_SY.tC_CB_ESL.Di			:=	IN_SY.tC_CB_ESL.Di			OR	NOT IN_SY.tC_CB_ESL.GoodQual;

	IN_SY.tLineCB_On.Di			:=	IN_SY.tLineCB_On.Di			OR	NOT IN_SY.tLineCB_On.GoodQual;

	IN_SY.tEngDemIsland.Di		:=	IN_SY.tEngDemIsland.Di		OR	NOT IN_SY.tEngDemIsland.GoodQual;
	(*------------------------------------------------------------------------------------*)

	IN_SY.tEarthCB_Off.Di		:=	IN_SY.tEarthCB_Off.Di		OR	NOT IN_SY.tEarthCB_Off.GoodQual;
	IN_SY.tIsoCB_Off.Di			:=	IN_SY.tIsoCB_Off.Di			OR	NOT IN_SY.tIsoCB_Off.GoodQual;
	IN_SY.tMnsOk_GTE.Di			:=	IN_SY.tMnsOk_GTE.Di			OR	NOT IN_SY.tMnsOk_GTE.GoodQual;
	IN_SY.tMnsOk_TGS.Di			:=	IN_SY.tMnsOk_TGS.Di			OR	NOT IN_SY.tMnsOk_TGS.GoodQual;
	IN_SY.tMnsOk_C13100.Di		:=	IN_SY.tMnsOk_C13100.Di		OR	NOT IN_SY.tMnsOk_C13100.GoodQual;

	IN_SY.tMCB_OpF_Ext.Di		:=	IN_SY.tMCB_OpF_Ext.Di		OR	NOT IN_SY.tMCB_OpF_Ext.GoodQual;
	IN_SY.tGCB_OpF_Ext.Di		:=	IN_SY.tGCB_OpF_Ext.Di		OR	NOT IN_SY.tGCB_OpF_Ext.GoodQual;
	(*------------------------------------------------------------------------------------*)

	IN_SY.tMnsOk_ClosCond_Ok.Di	:=	IN_SY.tMnsOk_ClosCond_Ok.Di	OR	NOT IN_SY.tMnsOk_ClosCond_Ok.GoodQual;
	IN_SY.tAfMnsF_ClosCond_Ok.Di := IN_SY.tAfMnsF_ClosCond_Ok.Di OR NOT IN_SY.tAfMnsF_ClosCond_Ok.GoodQual;

	IN_SY.tMidVoltCB_Failure.Di := IN_SY.tMidVoltCB_Failure.Di	OR NOT IN_SY.tMidVoltCB_Failure.GoodQual;
	IN_SY.tGndFault_BB.Di		:= IN_SY.tGndFault_BB.Di		OR NOT IN_SY.tGndFault_BB.GoodQual;

END_PROGRAM
```

### Program Logical/Synchronization/general_SY (IEC, version 4.12.0) - functions

#### general_SYCyclic.st
```iecst
(*******************************************************************************
general		general functions

This code is confidential and proprietary to the INNIO Company.
It may not be used in any form, or reproduced in any manner,
without the express written permission of the INNIO Company.
Copyright, INNIO Company, 2022

Customized modifications: -
------------------------

History:
-------
V3.90.0	17.10.2012	lettenb.	new
V3.99.0	07.03.2013	lettenb.	INIT: iEngNr added
		24.04.2013				changeover SyOMSS through status OFF added
V4.00.0	26.02.2014				OUT_SY.iIdx_SyOMSS FOR opstate added
V4.05.0 11.12.2017	lettenb.	check para setup added
		21.01.2018	Perktold,	hardware operation mode switch added
V4.07.1	23.07.2019	Denk,		Init: error handling for CfgGetIPAddr_ArWin.status added
V4.09.0	30.01.2020  lettenb.	bResetWarning added for gcbTC1
V4.10.0	25.02.2021	lettenb.	VIS2MM.iModule added(read IP-adr. not available for B&R IPC, removed), bugfix
V4.12.0	04.07.2022	lettenb.	OUT_SY.tSyOMSS_Man/Aut.Do added, dead bus synch

Instructions for use:
--------------------
Outstandings:
------------
*******************************************************************************)
PROGRAM _CYCLIC

	(* check para setup *)
	IN_SY.tPB2MM.bParaSetupOk;
	Para.iEng_Motortype;    (* MIN= 208   MAX= 920    *)
	Para.rN_EngStart_LimHi; (* MIN= 50.0  MAX= 2200.0 *)

	(* engine type defnition *)
	xEngType.Motortype := INT_TO_UINT(Para.iEng_Motortype);
	xEngType();				(* use: xEngType.Type2 as BOOL, ....*)

	(* engine operating mode selection *)
	bOMSS_Stop := FALSE;
	bOMSS_Man  := FALSE;
	bOMSS_Aut  := FALSE;
	bOMSS_Test := FALSE;
	bOMSS_Scav := FALSE;
	bOMSS_MAT  := FALSE;

	CASE IN_SY.iIdx_OMSS OF
	0:	bOMSS_Stop := TRUE;
	1:	bOMSS_Man  := TRUE;
		bOMSS_MAT  := TRUE;
	2:	bOMSS_Aut  := TRUE;
		bOMSS_MAT  := TRUE;
	3:	bOMSS_Test := TRUE;
		bOMSS_MAT  := TRUE;
	4:	bOMSS_Scav := TRUE;
	END_CASE;

	(* synchronization operating mode selection *)
	IF IN_SY.tHW_Switches.bGoodQual THEN
	(* HARDWARE OPERATION MODE SWITCHES *)
		OUT_SY.iIdx_SyOMSS	:= IN_SY.tHW_Switches.iIdx_SyOMS_Hw;

		xTON_SyOMSS_Man(IN:= OUT_SY.iIdx_SyOMSS = 1, PT:= T#200ms);
		xTON_SyOMSS_Aut(IN:= OUT_SY.iIdx_SyOMSS = 2, PT:= T#200ms);

		VIS2MM.iIdx_SyOMSS	:= INT_TO_DINT(OUT_SY.iIdx_SyOMSS);
	ELSE
	(* OPERATION MODE SWITCHES ON HMI *)
		OUT_SY.iIdx_SyOMSS := DINT_TO_INT(VIS2MM.iIdx_SyOMSS);

		xTON_SyOMSS_Man(IN:= VIS2MM.iIdx_SyOMSS = 1, PT:= T#200ms);
		xTON_SyOMSS_Aut(IN:= VIS2MM.iIdx_SyOMSS = 2, PT:= T#200ms);
	END_IF;

	bSyOMSS_Man :=     xTON_SyOMSS_Man.Q;
	bSyOMSS_Aut :=     xTON_SyOMSS_Aut.Q;
	bSyOMSS_Off := NOT bSyOMSS_Man AND NOT bSyOMSS_Aut;

	OUT_SY.tSyOMSS_Man.Do := bSyOMSS_Man;
	OUT_SY.tSyOMSS_Aut.Do := bSyOMSS_Aut;

	(* engine operating mode *)
	xOpMode(in:= IN_SY.iSt_OpMode);

	(* plc running *)
	IN_SY.tPB2MM.bSys_Run;

	(* reset *)
	bResetWarning := IN_SY.tAB2SY.bResetWarning;

	(*------------------------------------------------------------------------------------*)
	(* engine start speed limit *)
	xGR_MAXR_N_EngStart(In:= IN_SY.rN_EngAct, Gw:= Para.rN_EngStart_LimHi, Hy:= Para.rN_EngStart_HyHi);
	xTOF_N_EngStart(IN:= xGR_MAXR_N_EngStart.Q AND IN_SY.tPB2MM.bParaSetupOk, PT:= T#10s);
	bN_EngStart := xTOF_N_EngStart.Q;
	(*------------------------------------------------------------------------------------*)

	(* module number *)
	iEngNr := VIS2MM.iModule;
	OUT_SY.iModule := INT_TO_USINT(iEngNr);
END_PROGRAM
```

#### general_SYInit.st
```iecst
PROGRAM _INIT

END_PROGRAM
```

#### general_SY.var
```iecst
VAR
	xGR_MAXR_N_EngStart : GR_MAXR;
	xTOF_N_EngStart : TOF;
	xTON_SyOMSS_Man : TON;
	xTON_SyOMSS_Aut : TON;
END_VAR
```

### Program Logical/Synchronization/TBMode (IEC, version 4.13.0) - test bench mode

#### TBModeCyclic.st
```iecst
(*******************************************************************************
TbMode		test bench mode

This code is confidential and proprietary to the INNIO Company.
It may not be used in any form, or reproduced in any manner,
without the express written permission of the INNIO Company.
Copyright, INNIO Company, 2019

Customized modifications: -
------------------------

History:
-------
V3.99.0	26.02.2013	lettenb.	new
		19.11.2013				OUT_SY.bSmoothDischarge := FALSE; (IF OUT_SY.bTestBenchModeIsland) bugfix
V4.00.0 12.06.2014	lettenb.	test bTestBenchModeIsland
V4.03.0	14.08.2015	lettenb.	OUT_SY.bOnly_Island	logic for standard mode corr. removed (bugfix/pfanzagl)
V4.13.0	29.11.2023	Goenczi		SmoothDischarge set in CU module

Instructions for use:
--------------------
Outstandings:
------------
*******************************************************************************)
PROGRAM _CYCLIC

	(******************************************************************************)
	(* test-bench mode timeout control *)                        (* from settings *)

	xTON_PRF(IN:= IN_SY.tTBMode.Di, PT:= T#10s);
	xR_TRIG_PRF(CLK:= xTON_PRF.Q);

	IF NOT IN_SY.tTBMode.Di OR NOT IN_SY.tPB2MM.bSys_Run THEN
		xTOF_PRF(IN:= FALSE, PT:= T#0s);	(* reset timer *)
	ELSE
		xTOF_PRF(IN:= xR_TRIG_PRF.Q AND IN_SY.tPB2MM.bSys_Run, PT:= T#12h);
	END_IF;

	xTON_NP(IN:= IN_SY.tReq_PowMod.Di, PT:= T#10s);

	OUT_SY.bTestBenchModeIsland		:=	xTOF_PRF.Q
								AND NOT xTON_NP.Q
								AND NOT Para.bMCB_Enable
								AND NOT Para.bMCB_Ctr_Cust
								AND	   (IN_SY.tMCB_Off.Di OR NOT IN_SY.tMCB_Off.GoodQual)
								AND 	IN_SY.tC_CB_Off.Di;

	OUT_SY.bTestBenchModeParallel	:=	xTOF_PRF.Q
								AND     xTON_NP.Q
								AND NOT Para.bMCB_Enable
								AND NOT Para.bMCB_Ctr_Cust
								AND NOT Para.bMSy;

	bTestBenchMode	:=	OUT_SY.bTestBenchModeIsland OR OUT_SY.bTestBenchModeParallel;		(* test-bench mode *)

	(******************************************************************************)

	(*-----------------------------------------------------------------------------*)
	(* TestBenchMode - write in interfaces *)                      (* from pb17_en *)
	(*-----------------------------------------------------------------------------*)
	//	(* enable netp.operation for test-bench run *)
	IF	OUT_SY.bTestBenchModeParallel THEN
		IF	Para.bOnlyIsland_Enable THEN
			IN_SY.tMnsOk.Di	:=	OUT_SY.bMCB_On;
		END_IF;
	END_IF;

	(* switch standard-inputs esy to nonexisting required inputs esy *)
	IF OUT_SY.bTestBenchModeIsland THEN
		IF	Para.bMSy AND Para.bSyActive THEN
			IN_SY.tGCB_AGO.Di	:=	TRUE;		(* enable closing gcb for test-bench run *)
		END_IF;
	END_IF;

	(*-----------------------------------------------------------------------------*)
	(* TestBenchMode - write out interfaces *)                  (* from ex pb17_en *)
	(*-----------------------------------------------------------------------------*)
	IF        OUT_SY.bTestBenchModeIsland THEN
		OUT_SY.bMCB_On			:=  IN_SY.tMCB_On.Di AND IN_SY.tMnsOk.Di;	(* mcb closed for engine control and RPS *)
		OUT_SY.bSmoothDischarge	:=	FALSE;									(* smoothly discharging power in island operation *)

	ELSIF NOT OUT_SY.bTestBenchModeIsland THEN
		OUT_SY.bMCB_On			:=  IN_SY.tMCB_On.Di;
		OUT_SY.bSmoothDischarge	:=	IN_SY.bSmoothDischarge_CU;
	END_IF;

	IF OUT_SY.bTestBenchModeParallel THEN
		OUT_SY.bOnly_Island	:= FALSE;
	ELSE
		IF OUT_SY.bTestBenchModeIsland THEN
			OUT_SY.bOnly_Island	:= (Para.bOnlyIsland_Enable OR	Para.bMSy);	(* enable only isl. op. for test-bench run *)
		ELSE
			OUT_SY.bOnly_Island	:=  Para.bOnlyIsland_Enable					(* enable only isl. op. as standard mode *)
							  OR   (Para.bMSy AND IN_SY.tOnly_Island.Di);
		END_IF;
	END_IF;

	(*-----------------------------------------------------------------------------*)

END_PROGRAM
```

#### TBMode.var
```iecst
VAR
	xTON_PRF : TON;
	xR_TRIG_PRF : R_TRIG;
	xTON_NP : TON;
	xTOF_PRF : TOF;
END_VAR
```

### Program Logical/Synchronization/sy_in (IEC, version 4.13.0) - in signals handling

#### sy_inCyclic.st
```iecst
(*******************************************************************************
sy_in				Switch standard-inputs from DI to internal variables

This code is confidential and proprietary to the INNIO Company.
It may not be used in any form, or reproduced in any manner,
without written permission of the INNIO Company.
Copyright, INNIO Company, 2019

Customized modifications: -
------------------------

History:
-------
V2.12	24.04.2006	LH			adapted for esy new
		31.10.2006	LH			new: general release gcb from Para.bMSy
		11.11.2006	LH			revised after Para.bMSy test
		20.11.2006	LH			revised for final release esy new
V2.20	07.02.2007	LH			adapted for supporting customer mcb
								enable signals from customer at any time
		27.02.2007	LH			simulate AUEB2 for old hardware
V2.30	18.01.2008	LH			adapted for test-bench run
V2.60.0	12.08.2009	lettenb.	ton_ccb_psf added
								gcb[0].IN_SY.bOtherGenParallel added
V3.20.0	30.09.2010	maier (BuR)	IN_SY.tGCB_On.Di changed to bGCB_ON
					maier (BuR)	IN_SY.tGCB_On.Di replaced with IN_SY.tGCB_On.Di
		01.10.2010	maier (BuR) OUT_SY.bMCB_On changed to bMCB_ON
					maier (BuR) IN_SY.tMCB_On.Di replaced with OUT_SY.bMCB_On
V3.90.0	13.11.2012	lettenb.	parts from pb17_en included
V3.99.0	26.02.2013	lettenb.	cleanup
		19.04.2013				mcb.on, mcb.rdy: Para.bMCB_Enable removed, active for all variants
								mcb.off: OR (NOT Para.bMCB_Enable AND NOT IN_SY.tMCB_Off.GoodQual AND NOT mcb.on)
										 added, if only MCB_On.Di exists
		18.07.2013				mains.enable included from setting_SY(task removed)
		21.11.2013				gcb.all_other_gcb_off: bTestBenchModeIsland added
V4.00.0	12.06.2014 lettenb.		changes after bTestBenchModeIsland test
V4.00.1	25.06.2015 lettenb.		rel_mcb_on2d_bb, rel_gcb_on2d_bb: gcb.esl, gcb.edc -> ccb.esl, ccb.edc /bugfix
V4.03.0	01.10.2015 lettenb.		Para.bGCB_MainsCutOff_Active added(reqisition request)
V4.07.0 17.05.2019 lettenb.		version, comment
V4.10.0 15.10.2020 lettenb.		sel_gcb_mains_cut_off: MIF only active, when island is not released, bugfix
V4.13.0 29.11.2023 Goenczi		bGCB_OGP_Bus other genset paralell bit via bus

Instructions for use:
--------------------
Define variants, where marked.

Outstandings:
------------
comment variants
*******************************************************************************)

(*		basic configuration:
		--------------------

	                           mains
	                             |
	                            mcb
	                             |      bb
	                        +----+---------------+----+
	                             |               |
	                            gcb             ccb = customer cb(generator)
	                             |               |
	                             |               |
	                             G               G

---------------------------------------------------------------------------------------------

		V3.40			V3.99		variante:	+MCB			+CCB			GSy
										immer			ESy+Msy  		noSy			AB_Sy
---------------------------------------------------------------------------------------------
immer	DI_GCB_ON_TC1	tGCB_On
		DI_GCB_OFF		tGCB_Off
		DI_GCB_RDY		tGCB_Rdy
		DI_GCB_RAC		tGCB_Rac
		DI_GCB_OL_TC1	tGCB_OL
		DI_GCB_SM1		tGCB_SM1
		DI_GCB_SM2		tGCB_SM2

		DI_MNS_OK_TC1	tMnsOk
		DI_MNS_MDF		tMns_MDF

MCB		DI_MCB_ON_TC1	tMCB_On
		DI_MCB_OFF		tMCB_Off
		DI_MCB_RDY		tMCB_Rdy
		DI_MCB_RAC		tMCB_Rac
		DI_MCB_OL		tMCB_OL
		DI_MCB_REM		tMCB_Rem
		DI_MCB_SM		tMCB_SM

CCB		DI_C_CB_ON		tC_CB_On
		DI_C_CB_OFF		tC_CB_Off
		DI_C_CB_EDC		tC_CB_EDC
		DI_C_CB_ESL		tC_CB_ESL

msy		DI_ENG_DI		tEngDemIsland
		DI_ENG_D		IN_SY.bEng_RPSDem;
		DI_GCB_MDL		tGCB_MDL
		DI_GCB_MRC		tGCB_MRC
		DI_GCB_AGO		tGCB_AGO
		DI_GCB_RI		tGCB_RI
		DI_GCB_OGP		tGCB_OGP
		DI_GCB_DVM		IN_GC.tGCB_DVM	(used in MM_GC)
		DI_ONLY_ISL		tOnly_Island

no msy	DI_REL_I		tRel_I
		DI_REL_BS		tRel_BS

AB/SYonsite
		DI_GCB_DSY		tGCB_DSY
		SynchNH/L		tF_N_DI_Inc.Di/F_N_DI_Dec.Di
		DI_u_plus/minus	tU_Adj_Plus.Di/tU_Adj_Minus.Di
						tU_Gen_Inc.Di/tU_Gen_Dec.Di

option	DI_DMND_PM		tReq_PowMod
		LIN_EIN			tLineCB_On
		F_BLO			tRelEngOpFromGSy
		FRG_RS			tGCB_DRM
						IN_SY.bRelSyFromCU

engine	DO_SY_LFG		IN_SY.tRel_Sync_Load.Do;
		DI_IN_RDY		IN_SY.bEng_Rdy_Aut_Exc;

*)
PROGRAM _CYCLIC
	(*-----------------------------------------------------------------------------*)
	(* reset gcb/mcb on/off button from vis *)
	IF bGCB_MOn THEN VIS2MM.bGCB_MOn := FALSE;	END_IF;
	IF bGCB_MOf THEN VIS2MM.bGCB_MOf := FALSE;	END_IF;

	bGCB_MOn := VIS2MM.bGCB_MOn;
	bGCB_MOf := VIS2MM.bGCB_MOf;

	IF bMCB_MOn THEN VIS2MM.bMCB_MOn := FALSE;	END_IF;
	IF bMCB_MOf THEN VIS2MM.bMCB_MOf := FALSE;	END_IF;

	bMCB_MOn := VIS2MM.bMCB_MOn;
	bMCB_MOf := VIS2MM.bMCB_MOf;

	(*-----------------------------------------------------------------------------*)
	IF	Para.bSyActive	THEN
		IF	IN_SY.tGCB_AGO.Di AND (IN_SY.tGCB_OGP.Di OR IN_SY.bGCB_OGP_Bus) THEN
			IN_SY.tGCB_AGO.Di	:=	FALSE;				(* MSY other gcb on *)
		END_IF;
	END_IF;

	IF	NOT Para.bSyActive	THEN
		gcb.on	:= IN_SY.tGCB_On.Di;					(* for onsite SY *)
	END_IF;

	(*----------------------------------------------------------------------------*)
	(*----------------------------------------------------------------------------*)
	mains.enable			:=	Para.bMns_Enable	(* enable mains = IN_SY.tMnsOk.Di existing*)
							OR	Para.bMSy
							OR	Para.bMCB_Ctr_Cust
							OR	OUT_SY.bTestBenchModeParallel;

	sel_gcb_mains_cut_off	:= (Para.bBS_OnlyMan OR	(Para.bMIF_Enable AND NOT IN_SY.tGCB_RI.Di) OR Para.bGCB_MainsCutOff_Active)
						AND NOT Para.bMSy;

	(*----------------------------------------------------------------------------*)

	IF	Para.bSyActive	THEN

		(* general -------------------------------------------------------------------*)
		bb_alive	:=      IN_SY.tBB_Alive.Di	(* busbar alive = voltage high *)
					OR (NOT IN_SY.tBB_Dead_MMD[1].Di AND IN_SY.tBB_Dead_MMD[1].GoodQual);

		IN_SY.tRel_I.Di;								(* release island/isolated operation *)
		IN_SY.tRel_BS.Di;								(* release black-out start   *)
		IN_SY.tRel_LS.Di;								(* load shedd ok = load shedding is done *)

		(* generator circuit breaker -------------------------------------------------*)
		gcb.eng_run				:=		bN_EngStart; 										(* engine rotating *)	//A_DREHZ;
		gcb.eng_oper			:=		IN_SY.tEng_Run.Do;									(* engine operation *)	//BTRB;
		gcb.eng_demanded 		:=		IN_SY.bEng_RPSDem; 									(* engine demanded *)	//A_AGFD;
		gcb.racked_in 			:=		IN_SY.tGCB_Rac.Di;									(* gcb racked in *)

		xTOF_gcb_rdy(IN:= IN_SY.tGCB_Rdy.Di, PT:= T#500ms);
		gcb.rdy					:=		xTOF_gcb_rdy.Q		AND		gcb.racked_in;			(* gcb ready for closing *)
		gcb.on					:=		IN_SY.tGCB_On.Di	AND		gcb.racked_in;			(* gcb closed *)
		gcb.off					:=		IN_SY.tGCB_Off.Di	OR	NOT gcb.racked_in;			(* gcb open *)
		gcb.man_off				:=		bGCB_MOf; 											(* gcb manual off command button *)
		gcb.man_on				:=		bGCB_MOn; 											(* gcb manual on  command button *)
		gcb.mdl					:=		IN_SY.tGCB_MDL.Di;									(* Para.bMSy *)
		gcb.mrc					:=		IN_SY.tGCB_MRC.Di 	OR OUT_SY.bTestBenchModeIsland;	(* Para.bMSy *)
		gcb.rel_island			:= 	   (IN_SY.tGCB_RI.Di  	OR OUT_SY.bTestBenchModeIsland)	AND	NOT	OUT_SY.bTestBenchModeParallel;	(* Para.bMSy *)
		gcb.all_other_gcb_off	:=		IN_SY.tGCB_AGO.Di	OR OUT_SY.bTestBenchModeIsland;
		gcb.other_gcb_on 		:=	NOT gcb.all_other_gcb_off;
		gcb.other_gen_parallel  :=		IN_SY.tGCB_OGP.Di OR IN_SY.bGCB_OGP_Bus;

		(* mains ---------------------------------------------------------------------*)
		mains.ok		:=		mains.enable	AND		IN_SY.tMnsOk.Di;				(* mains ok *)

		(* mains circuit breaker -----------------------------------------------------*)
		mcb.racked_in 	:=		IN_SY.tMCB_Rac.Di;										(* mcb racked in *)

		xTOF_mcb_rdy(IN:= IN_SY.tMCB_Rdy.Di, PT:= T#500ms);
		mcb.rdy			:=		xTOF_mcb_rdy.Q   AND mcb.racked_in;(* mcb ready for closing *)
		mcb.on			:=		IN_SY.tMCB_On.Di AND mcb.racked_in;(* mcb closed *)

		IF Para.bMSy OR OUT_SY.bTestBenchModeIsland THEN
			mcb.off		:=	   (Para.bIslandOp_Enable OR Para.bOnlyIsland_Enable OR Para.bMSy OR OUT_SY.bTestBenchModeIsland)
						AND	NOT	Para.bMCB_Ctr_Cust										(* mcb opened simulated (MSy) *)
						AND NOT	mcb.on;
		ELSE
			mcb.off		:= (NOT	Para.bMCB_Enable AND NOT Para.bIslandOp_Enable AND NOT Para.bOnlyIsland_Enable AND NOT Para.bMSy AND NOT Para.bMCB_Ctr_Cust)
						OR (NOT Para.bMCB_Enable AND NOT IN_SY.tMCB_Off.GoodQual AND NOT mcb.on)
						OR		IN_SY.tMCB_Off.Di
						OR	NOT	mcb.racked_in;											(* mcb opened from input *)
		END_IF;

		mcb.remote		:=		IN_SY.tMCB_Rem.Di;										(* mcb operation mode remote *)
		mcb.man_off		:=		bMCB_MOf 			AND 	Para.bMCB_Enable;			(* mcb manual off command *)
		mcb.man_on		:=		bMCB_MOn 			AND 	Para.bMCB_Enable;			(* mcb manual on command *)

		(* customer circuit breaker/external unit  -------------------------------------------------------------*)
		IF Para.bMSy THEN
			ccb.eng_demanded 		:=	FALSE;											(* external engine demanded *)
			ccb.eng_run				:=	FALSE;											(* external engine running  *)
			ccb.eng_oper			:=	FALSE;											(* external engine operation *)
			ccb.on					:=	FALSE;											(* external cb closed *)
			ccb.off					:=	TRUE;											(* external cb open *)
			ccb.alm_psf				:=	FALSE;											(* external cb position signal failure *)
			ccb.opf					:=	FALSE;											(* external cb opening failure *)
			ccb.esl					:=	FALSE;											(* external cb locked *)
			ccb.edc_in				:=	FALSE;											(* external cb demand closing to dead busbar *)
			ccb.other_gen_parallel  :=	FALSE;											(* external cb other gen parallel *)

		ELSE
			ccb.eng_demanded 		:=	IN_SY.tC_CB_On.Di OR FALSE;						(* external engine demanded *)
			ccb.eng_run				:=	IN_SY.tC_CB_On.Di;								(* external engine running  *)

			xTON_c_eng_op(IN:= ccb.eng_run, PT:= T#0s);

			ccb.eng_oper			:=	xTON_c_eng_op.Q;								(* external engine operating *)
			ccb.on					:=	IN_SY.tC_CB_On.Di;								(* external cb closed *)
			ccb.off					:=	IN_SY.tC_CB_Off.Di	OR	NOT	Para.bC_CB_Enable;	(* external cb open *)

			xTON_ccb_psf(IN:=   (	ccb.on	AND		ccb.off)
					 		OR (NOT ccb.on	AND	NOT ccb.off), PT:= T#3s);

			ccb.alm_psf				:=	xTON_ccb_psf.Q AND Para.bC_CB_Enable;			(* external cb position signal failure *)
			ccb.opf					:=	FALSE AND Para.bC_CB_Enable;					(* external cb opening failure, set TRUE if signal available *)
			ccb.esl					:=	IN_SY.tC_CB_ESL.Di;								(* external cb locked *)
			ccb.edc_in				:=	IN_SY.tC_CB_EDC.Di;								(* external cb demand closing to dead busbar *)
			ccb.other_gen_parallel  :=	FALSE AND Para.bC_CB_Enable;					(* external cb other gen parallel, set TRUE if signal available *)
		END_IF;

		(*----------------------------------------------------------------------------*)
		(* external unit demand lock gcb *)		(* ANF_BLO *)
		ccb.edc 		:=	Para.bC_CB_Enable		(* demand close from external gcb *)
					AND		bb_dead
					AND		ccb.edc_in;

		any_gcb_edc_bb	:=	ccb.edc;

		(*----------------------------------------------------------------------------*)
		(* MSY/external unit status cb locked 	(FRG_AES) *)
		(* release closing mcb to dead busbar *)
		rel_mcb_on2d_bb	:= (NOT Para.bC_CB_Enable AND NOT Para.bMCB_Ctr_Cust) OR (ccb.esl AND NOT ccb.edc);

		(* release closing gcb to dead busbar *)
		rel_gcb_on2d_bb :=((NOT Para.bC_CB_Enable AND NOT Para.bMCB_Ctr_Cust) OR (ccb.esl AND NOT ccb.edc))
						AND		gcb.mrc				(* release closing from MSy *)
						AND	NOT	gcb.mdl;			(* no lock from MSy         *)

		(*----------------------------------------------------------------------------*)
	END_IF;

END_PROGRAM
```

#### sy_in.var
```iecst
VAR
	xTOF_gcb_rdy : TOF;
	xTOF_mcb_rdy : TOF;
	xTON_c_eng_op : TON;
	xTON_ccb_psf : TON;
END_VAR
```

### Program Logical/Synchronization/MsgSY (IEC, version 4.14.0) - messages
